// TwinCAT 3 PLC project PLC_MR
// ProgramVersion: 3.1.4026.16
// libraries:
//   Tc2_ControllerToolbox, * (Beckhoff Automation GmbH)
//   Tc2_SerialCom, * (Beckhoff Automation GmbH)
//   Tc2_Standard, * (Beckhoff Automation GmbH)
//   Tc2_System, * (Beckhoff Automation GmbH)
//   Tc2_Utilities, * (Beckhoff Automation GmbH)
//   Tc3_BA_Common, * (Beckhoff Automation GmbH)
//   Tc3_Module, * (Beckhoff Automation GmbH)
// project tree:
//   DUTs/ E_ControlMode.TcDUT, E_RampGeneratorState.TcDUT, E_RecipeRunETMode.TcDUT, E_RecipeRun.TcDUT, E_TowerLamp.TcDUT, OperationMode.TcDUT, outWord.TcDUT, RampGeneratorInput.TcDUT, RecipeRunET.TcDUT, RecipeStep.TcDUT, ScaleFactor.TcDUT (not stored)
//   FUNTION/ BOOL_TO_STRING_LHeaterON.TcPOU (not stored), CheckRangeSigned.TcPOU (not stored), CheckRangeUnsigned.TcPOU, HEXSTR_TO_REAL_LHeaterPV.TcPOU (not stored), Real_To_String_LineHeater.TcPOU, Real_To_String_ThermalBath.TcPOU, USINT_TO_WORD_Bit.TcPOU, WORD_TO_USINT_Bit.TcPOU
//   GVLs/ GVL_IO.TcGVL, GVL_Serial.TcGVL, RCP.TcGVL
//   / PlcTask.TcTTO (not stored), PlcTask_Standard.TcTTO
//   POUs/ FB_AnalogDeviceRampControl.TcPOU, FB_ControlRampGenerator.TcPOU, FB_DeviationCheck.TcPOU, FB_FaultCheck.TcPOU, FB_OverLimitCheck.TcPOU, FB_RecipeAnalogControlInputSequencer.TcPOU, FB_SensorLimitCheck.TcPOU, FB_TON_Pausable.TcPOU, FB_ValveControl.TcPOU, F_ResetTimersAndRCPTimes.TcPOU, MAIN.TcPOU, P11_E3508.TcPOU, P12_IQ_PLUS.TcPOU, P13_LineHeater.TcPOU, P14_ThermalBath.TcPOU, P15_RotationOperation.TcPOU, P16_CoverOperation.TcPOU, P17_DOROperation.TcPOU, P20_BackgroundCom.TcPOU (not stored), P21_Background_LineHeater.TcPOU, P22_Background_ThermalBath.TcPOU (not stored), P30_ManualControl.TcPOU, P50_RecipeControl.TcPOU, P60_UpdatePV.TcPOU, P70_Interface.TcPOU, P90_Interlock.TcPOU, P91_Monitoring.TcPOU, P92_Maintenance.TcPOU, P31_PriorityControl.TcPOU
// real-time tasks:
//   TASK PlcTask_Standard: cycle T#10ms, priority 21, ADS port 350
//   TASK PlcTask: cycle T#2ms, priority 19, ADS port 351
// I/O:
//   DEVICE Device 1 (EtherCAT) (disabled), AmsNetId 211.225.0.130.2.1
//     Term 1 (EK1200) [EK1200-5000 EtherCAT Power supply (2A E-Bus)]
//       Term 2 (EL6752) [EL6752 DeviceNet Master]
//       Term 3 (EL9011) [EL9011 End Terminal]
//   DEVICE Device 2 (EL6752) (disabled), AmsNetId 10.10.10.10.3.1
//     Box 1  (BK5220) // Bus Coupler
//     Box 2  (BK5220) // Bus Coupler
//     N4E0 1 // EDS-File: 'OPP6-2D.eds' DescText: OPP6-2D Vendor: CKD Corporation Device Type: Generic Device Product Name: OPP6-2D Catalog Number:
//     N4E0 2 // EDS-File: 'OPP6-2D.eds' DescText: OPP6-2D Vendor: CKD Corporation Device Type: Generic Device Product Name: OPP6-2D Catalog Number:
//     IQ-Plus // EDS-File: 'TBJQPDNG-L041X01 155Out154.eds' DescText: Intellisys IQ-Plus Vendor: Nor-Cal Products Device Type: Process Control Valve Product Name: INTELLISYS Catalog Number: IQ-Plus
//     E3508 // EDS-File: '3500-3.eds' DescText: Eurotherm 3500 Vendor: Eurotherm Device Type: Generic Product Name: Eurotherm 3500 Catalog Number:
//   DEVICE Device 3 (NOV-DP-RAM) (disabled)
// variable links:
//   PLC_MR/PLC_MR Instance <-> Device 2 (EL6752)/Box 1  (BK5220)
//     PlcTask_Standard Inputs/GVL_IO.aAnalogInputIO[1] <-> Term 15 (KL3464)/Channel 1/MFC01
//     PlcTask_Standard Inputs/GVL_IO.aAnalogInputIO[2] <-> Term 15 (KL3464)/Channel 2/MFC02
//     PlcTask_Standard Inputs/GVL_IO.aAnalogInputIO[3] <-> Term 15 (KL3464)/Channel 3/MFC03
//     PlcTask_Standard Inputs/GVL_IO.aAnalogInputIO[4] <-> Term 15 (KL3464)/Channel 4/MFC04
//     PlcTask_Standard Inputs/GVL_IO.aAnalogInputIO[5] <-> Term 17 (KL3464)/Channel 1/MFC05
//     PlcTask_Standard Inputs/GVL_IO.aAnalogInputIO[6] <-> Term 17 (KL3464)/Channel 2/MFC06
//     PlcTask_Standard Inputs/GVL_IO.aAnalogInputIO[7] <-> Term 17 (KL3464)/Channel 3/MFC07
//     PlcTask_Standard Inputs/GVL_IO.aAnalogInputIO[8] <-> Term 17 (KL3464)/Channel 4/MFC08
//     PlcTask_Standard Inputs/GVL_IO.aDigitalInputIO[{1..9}] <-> Term {2..10} (KL1408)/Channel 1/Input  (9 links)
//     PlcTask_Standard Inputs/GVL_IO.aDigitalInputIO[1] @bit 1 <-> Term 2 (KL1408)/Channel 2/Input
//     PlcTask_Standard Inputs/GVL_IO.aDigitalInputIO[1] @bit 2 <-> Term 2 (KL1408)/Channel 3/Input
//     PlcTask_Standard Inputs/GVL_IO.aDigitalInputIO[1] @bit 3 <-> Term 2 (KL1408)/Channel 4/Input
//     PlcTask_Standard Inputs/GVL_IO.aDigitalInputIO[1] @bit 4 <-> Term 2 (KL1408)/Channel 5/Input
//     PlcTask_Standard Inputs/GVL_IO.aDigitalInputIO[1] @bit 5 <-> Term 2 (KL1408)/Channel 6/Input
//     PlcTask_Standard Inputs/GVL_IO.aDigitalInputIO[1] @bit 6 <-> Term 2 (KL1408)/Channel 7/Input
//     PlcTask_Standard Inputs/GVL_IO.aDigitalInputIO[1] @bit 7 <-> Term 2 (KL1408)/Channel 8/Input
//     PlcTask_Standard Inputs/GVL_IO.aDigitalInputIO[2] @bit 1 <-> Term 3 (KL1408)/Channel 2/Input
//     PlcTask_Standard Inputs/GVL_IO.aDigitalInputIO[2] @bit 2 <-> Term 3 (KL1408)/Channel 3/Input
//     PlcTask_Standard Inputs/GVL_IO.aDigitalInputIO[2] @bit 3 <-> Term 3 (KL1408)/Channel 4/Input
//     PlcTask_Standard Inputs/GVL_IO.aDigitalInputIO[2] @bit 4 <-> Term 3 (KL1408)/Channel 5/Input
//     PlcTask_Standard Inputs/GVL_IO.aDigitalInputIO[2] @bit 5 <-> Term 3 (KL1408)/Channel 6/Input
//     PlcTask_Standard Inputs/GVL_IO.aDigitalInputIO[2] @bit 6 <-> Term 3 (KL1408)/Channel 7/Input
//     PlcTask_Standard Inputs/GVL_IO.aDigitalInputIO[2] @bit 7 <-> Term 3 (KL1408)/Channel 8/Input
//     PlcTask_Standard Inputs/GVL_IO.aDigitalInputIO[3] @bit 1 <-> Term 4 (KL1408)/Channel 2/Input
//     PlcTask_Standard Inputs/GVL_IO.aDigitalInputIO[3] @bit 2 <-> Term 4 (KL1408)/Channel 3/Input
//     PlcTask_Standard Inputs/GVL_IO.aDigitalInputIO[3] @bit 3 <-> Term 4 (KL1408)/Channel 4/Input
//     PlcTask_Standard Inputs/GVL_IO.aDigitalInputIO[3] @bit 4 <-> Term 4 (KL1408)/Channel 5/Input
//     PlcTask_Standard Inputs/GVL_IO.aDigitalInputIO[3] @bit 5 <-> Term 4 (KL1408)/Channel 6/Input
//     PlcTask_Standard Inputs/GVL_IO.aDigitalInputIO[3] @bit 6 <-> Term 4 (KL1408)/Channel 7/Input
//     PlcTask_Standard Inputs/GVL_IO.aDigitalInputIO[3] @bit 7 <-> Term 4 (KL1408)/Channel 8/Input
//     PlcTask_Standard Inputs/GVL_IO.aDigitalInputIO[4] @bit 1 <-> Term 5 (KL1408)/Channel 2/Input
//     PlcTask_Standard Inputs/GVL_IO.aDigitalInputIO[4] @bit 2 <-> Term 5 (KL1408)/Channel 3/Input
//     PlcTask_Standard Inputs/GVL_IO.aDigitalInputIO[4] @bit 3 <-> Term 5 (KL1408)/Channel 4/Input
//     PlcTask_Standard Inputs/GVL_IO.aDigitalInputIO[4] @bit 4 <-> Term 5 (KL1408)/Channel 5/Input
//     PlcTask_Standard Inputs/GVL_IO.aDigitalInputIO[4] @bit 5 <-> Term 5 (KL1408)/Channel 6/Input
//     PlcTask_Standard Inputs/GVL_IO.aDigitalInputIO[4] @bit 6 <-> Term 5 (KL1408)/Channel 7/Input
//     PlcTask_Standard Inputs/GVL_IO.aDigitalInputIO[4] @bit 7 <-> Term 5 (KL1408)/Channel 8/Input
//     PlcTask_Standard Inputs/GVL_IO.aDigitalInputIO[5] @bit 1 <-> Term 6 (KL1408)/Channel 2/Input
//     PlcTask_Standard Inputs/GVL_IO.aDigitalInputIO[5] @bit 2 <-> Term 6 (KL1408)/Channel 3/Input
//     PlcTask_Standard Inputs/GVL_IO.aDigitalInputIO[5] @bit 3 <-> Term 6 (KL1408)/Channel 4/Input
//     PlcTask_Standard Inputs/GVL_IO.aDigitalInputIO[5] @bit 4 <-> Term 6 (KL1408)/Channel 5/Input
//     PlcTask_Standard Inputs/GVL_IO.aDigitalInputIO[5] @bit 5 <-> Term 6 (KL1408)/Channel 6/Input
//     PlcTask_Standard Inputs/GVL_IO.aDigitalInputIO[5] @bit 6 <-> Term 6 (KL1408)/Channel 7/Input
//     PlcTask_Standard Inputs/GVL_IO.aDigitalInputIO[5] @bit 7 <-> Term 6 (KL1408)/Channel 8/Input
//     PlcTask_Standard Inputs/GVL_IO.aDigitalInputIO[6] @bit 1 <-> Term 7 (KL1408)/Channel 2/Input
//     PlcTask_Standard Inputs/GVL_IO.aDigitalInputIO[6] @bit 2 <-> Term 7 (KL1408)/Channel 3/Input
//     PlcTask_Standard Inputs/GVL_IO.aDigitalInputIO[6] @bit 3 <-> Term 7 (KL1408)/Channel 4/Input
//     PlcTask_Standard Inputs/GVL_IO.aDigitalInputIO[6] @bit 4 <-> Term 7 (KL1408)/Channel 5/Input
//     PlcTask_Standard Inputs/GVL_IO.aDigitalInputIO[6] @bit 5 <-> Term 7 (KL1408)/Channel 6/Input
//     PlcTask_Standard Inputs/GVL_IO.aDigitalInputIO[6] @bit 6 <-> Term 7 (KL1408)/Channel 7/Input
//     PlcTask_Standard Inputs/GVL_IO.aDigitalInputIO[6] @bit 7 <-> Term 7 (KL1408)/Channel 8/Input
//     PlcTask_Standard Inputs/GVL_IO.aDigitalInputIO[7] @bit 1 <-> Term 8 (KL1408)/Channel 2/Input
//     PlcTask_Standard Inputs/GVL_IO.aDigitalInputIO[7] @bit 2 <-> Term 8 (KL1408)/Channel 3/Input
//     PlcTask_Standard Inputs/GVL_IO.aDigitalInputIO[7] @bit 3 <-> Term 8 (KL1408)/Channel 4/Input
//     PlcTask_Standard Inputs/GVL_IO.aDigitalInputIO[7] @bit 4 <-> Term 8 (KL1408)/Channel 5/Input
//     PlcTask_Standard Inputs/GVL_IO.aDigitalInputIO[7] @bit 5 <-> Term 8 (KL1408)/Channel 6/Input
//     PlcTask_Standard Inputs/GVL_IO.aDigitalInputIO[7] @bit 6 <-> Term 8 (KL1408)/Channel 7/Input
//     PlcTask_Standard Inputs/GVL_IO.aDigitalInputIO[7] @bit 7 <-> Term 8 (KL1408)/Channel 8/Input
//     PlcTask_Standard Inputs/GVL_IO.aDigitalInputIO[8] @bit 1 <-> Term 9 (KL1408)/Channel 2/Input
//     PlcTask_Standard Inputs/GVL_IO.aDigitalInputIO[8] @bit 2 <-> Term 9 (KL1408)/Channel 3/Input
//     PlcTask_Standard Inputs/GVL_IO.aDigitalInputIO[8] @bit 3 <-> Term 9 (KL1408)/Channel 4/Input
//     PlcTask_Standard Inputs/GVL_IO.aDigitalInputIO[8] @bit 4 <-> Term 9 (KL1408)/Channel 5/Input
//     PlcTask_Standard Inputs/GVL_IO.aDigitalInputIO[8] @bit 5 <-> Term 9 (KL1408)/Channel 6/Input
//     PlcTask_Standard Inputs/GVL_IO.aDigitalInputIO[8] @bit 6 <-> Term 9 (KL1408)/Channel 7/Input
//     PlcTask_Standard Inputs/GVL_IO.aDigitalInputIO[8] @bit 7 <-> Term 9 (KL1408)/Channel 8/Input
//     PlcTask_Standard Inputs/GVL_IO.aDigitalInputIO[9] @bit 1 <-> Term 10 (KL1408)/Channel 2/Input
//     PlcTask_Standard Inputs/GVL_IO.aDigitalInputIO[9] @bit 2 <-> Term 10 (KL1408)/Channel 3/Input
//     PlcTask_Standard Inputs/GVL_IO.aDigitalInputIO[9] @bit 3 <-> Term 10 (KL1408)/Channel 4/Input
//     PlcTask_Standard Inputs/GVL_IO.aDigitalInputIO[9] @bit 4 <-> Term 10 (KL1408)/Channel 5/Input
//     PlcTask_Standard Inputs/GVL_IO.aDigitalInputIO[9] @bit 5 <-> Term 10 (KL1408)/Channel 6/Input
//     PlcTask_Standard Inputs/GVL_IO.aDigitalInputIO[9] @bit 6 <-> Term 10 (KL1408)/Channel 7/Input
//     PlcTask_Standard Inputs/GVL_IO.aDigitalInputIO[9] @bit 7 <-> Term 10 (KL1408)/Channel 8/Input
//     PlcTask_Standard Outputs/GVL_IO.aAnalogOutputIO[1] <-> Term 16 (KL4404)/Channel 1/MFC01
//     PlcTask_Standard Outputs/GVL_IO.aAnalogOutputIO[2] <-> Term 16 (KL4404)/Channel 2/MFC02
//     PlcTask_Standard Outputs/GVL_IO.aAnalogOutputIO[3] <-> Term 16 (KL4404)/Channel 3/MFC03
//     PlcTask_Standard Outputs/GVL_IO.aAnalogOutputIO[4] <-> Term 16 (KL4404)/Channel 4/MFC04
//     PlcTask_Standard Outputs/GVL_IO.aAnalogOutputIO[5] <-> Term 18 (KL4404)/Channel 1/MFC05
//     PlcTask_Standard Outputs/GVL_IO.aAnalogOutputIO[6] <-> Term 18 (KL4404)/Channel 2/MFC06
//     PlcTask_Standard Outputs/GVL_IO.aAnalogOutputIO[7] <-> Term 18 (KL4404)/Channel 3/MFC07
//     PlcTask_Standard Outputs/GVL_IO.aAnalogOutputIO[8] <-> Term 18 (KL4404)/Channel 4/MFC08
//     PlcTask_Standard Outputs/GVL_IO.aDigitalOutputIO[{1..4}] <-> Term {11..14} (KL2408)/Channel 1/Output  (4 links)
//     PlcTask_Standard Outputs/GVL_IO.aDigitalOutputIO[1] @bit 1 <-> Term 11 (KL2408)/Channel 2/Output
//     PlcTask_Standard Outputs/GVL_IO.aDigitalOutputIO[1] @bit 2 <-> Term 11 (KL2408)/Channel 3/Output
//     PlcTask_Standard Outputs/GVL_IO.aDigitalOutputIO[1] @bit 3 <-> Term 11 (KL2408)/Channel 4/Output
//     PlcTask_Standard Outputs/GVL_IO.aDigitalOutputIO[1] @bit 4 <-> Term 11 (KL2408)/Channel 5/Output
//     PlcTask_Standard Outputs/GVL_IO.aDigitalOutputIO[1] @bit 5 <-> Term 11 (KL2408)/Channel 6/Output
//     PlcTask_Standard Outputs/GVL_IO.aDigitalOutputIO[1] @bit 6 <-> Term 11 (KL2408)/Channel 7/Output
//     PlcTask_Standard Outputs/GVL_IO.aDigitalOutputIO[1] @bit 7 <-> Term 11 (KL2408)/Channel 8/Output
//     PlcTask_Standard Outputs/GVL_IO.aDigitalOutputIO[2] @bit 1 <-> Term 12 (KL2408)/Channel 2/Output
//     PlcTask_Standard Outputs/GVL_IO.aDigitalOutputIO[2] @bit 2 <-> Term 12 (KL2408)/Channel 3/Output
//     PlcTask_Standard Outputs/GVL_IO.aDigitalOutputIO[2] @bit 3 <-> Term 12 (KL2408)/Channel 4/Output
//     PlcTask_Standard Outputs/GVL_IO.aDigitalOutputIO[2] @bit 4 <-> Term 12 (KL2408)/Channel 5/Output
//     PlcTask_Standard Outputs/GVL_IO.aDigitalOutputIO[2] @bit 5 <-> Term 12 (KL2408)/Channel 6/Output
//     PlcTask_Standard Outputs/GVL_IO.aDigitalOutputIO[2] @bit 6 <-> Term 12 (KL2408)/Channel 7/Output
//     PlcTask_Standard Outputs/GVL_IO.aDigitalOutputIO[2] @bit 7 <-> Term 12 (KL2408)/Channel 8/Output
//     PlcTask_Standard Outputs/GVL_IO.aDigitalOutputIO[3] @bit 1 <-> Term 13 (KL2408)/Channel 2/Output
//     PlcTask_Standard Outputs/GVL_IO.aDigitalOutputIO[3] @bit 2 <-> Term 13 (KL2408)/Channel 3/Output
//     PlcTask_Standard Outputs/GVL_IO.aDigitalOutputIO[3] @bit 3 <-> Term 13 (KL2408)/Channel 4/Output
//     PlcTask_Standard Outputs/GVL_IO.aDigitalOutputIO[3] @bit 4 <-> Term 13 (KL2408)/Channel 5/Output
//     PlcTask_Standard Outputs/GVL_IO.aDigitalOutputIO[3] @bit 5 <-> Term 13 (KL2408)/Channel 6/Output
//     PlcTask_Standard Outputs/GVL_IO.aDigitalOutputIO[3] @bit 6 <-> Term 13 (KL2408)/Channel 7/Output
//     PlcTask_Standard Outputs/GVL_IO.aDigitalOutputIO[3] @bit 7 <-> Term 13 (KL2408)/Channel 8/Output
//     PlcTask_Standard Outputs/GVL_IO.aDigitalOutputIO[4] @bit 1 <-> Term 14 (KL2408)/Channel 2/Output
//     PlcTask_Standard Outputs/GVL_IO.aDigitalOutputIO[4] @bit 2 <-> Term 14 (KL2408)/Channel 3/Output
//     PlcTask_Standard Outputs/GVL_IO.aDigitalOutputIO[4] @bit 3 <-> Term 14 (KL2408)/Channel 4/Output
//     PlcTask_Standard Outputs/GVL_IO.aDigitalOutputIO[4] @bit 4 <-> Term 14 (KL2408)/Channel 5/Output
//     PlcTask_Standard Outputs/GVL_IO.aDigitalOutputIO[4] @bit 5 <-> Term 14 (KL2408)/Channel 6/Output
//     PlcTask_Standard Outputs/GVL_IO.aDigitalOutputIO[4] @bit 6 <-> Term 14 (KL2408)/Channel 7/Output
//     PlcTask_Standard Outputs/GVL_IO.aDigitalOutputIO[4] @bit 7 <-> Term 14 (KL2408)/Channel 8/Output
//   PLC_MR/PLC_MR Instance <-> Device 2 (EL6752)/Box 2  (BK5220)
//     PlcTask Inputs/P21_Background_LineHeater.stIn_KL6031_LH/D <-> Term 34 (KL6031)/Channel 1/Data In 0
//     PlcTask Inputs/P21_Background_LineHeater.stIn_KL6031_LH/D @bit {8..168 step 8} <-> Term 34 (KL6031)/Channel 1/Data In {1..21}  (21 links)
//     PlcTask Inputs/P21_Background_LineHeater.stIn_KL6031_LH/Status <-> Term 34 (KL6031)/Channel 1/State
//     PlcTask Inputs/P22_Background_ThermalBath.stIn_KL6031_TB/D <-> Term 35 (KL6031)/Channel 1/Data In 0
//     PlcTask Inputs/P22_Background_ThermalBath.stIn_KL6031_TB/D @bit {8..168 step 8} <-> Term 35 (KL6031)/Channel 1/Data In {1..21}  (21 links)
//     PlcTask Inputs/P22_Background_ThermalBath.stIn_KL6031_TB/Status <-> Term 35 (KL6031)/Channel 1/State
//     PlcTask Outputs/P21_Background_LineHeater.stOut_KL6031_LH/Ctrl <-> Term 34 (KL6031)/Channel 1/Ctrl
//     PlcTask Outputs/P21_Background_LineHeater.stOut_KL6031_LH/D <-> Term 34 (KL6031)/Channel 1/Data Out 0
//     PlcTask Outputs/P21_Background_LineHeater.stOut_KL6031_LH/D @bit {8..168 step 8} <-> Term 34 (KL6031)/Channel 1/Data Out {1..21}  (21 links)
//     PlcTask Outputs/P22_Background_ThermalBath.stOut_KL6031_TB/Ctrl <-> Term 35 (KL6031)/Channel 1/Ctrl
//     PlcTask Outputs/P22_Background_ThermalBath.stOut_KL6031_TB/D <-> Term 35 (KL6031)/Channel 1/Data Out 0
//     PlcTask Outputs/P22_Background_ThermalBath.stOut_KL6031_TB/D @bit {8..168 step 8} <-> Term 35 (KL6031)/Channel 1/Data Out {1..21}  (21 links)
//     PlcTask_Standard Inputs/GVL_IO.aAnalogInputIO2[1] <-> Term 32 (KL3152)/Channel 1/RotaionPV
//     PlcTask_Standard Inputs/GVL_IO.aAnalogInputIO[10] <-> Term 20 (KL3464)/Channel 2/MFC10
//     PlcTask_Standard Inputs/GVL_IO.aAnalogInputIO[11] <-> Term 20 (KL3464)/Channel 3/MFC11
//     PlcTask_Standard Inputs/GVL_IO.aAnalogInputIO[12] <-> Term 20 (KL3464)/Channel 4/MFC12
//     PlcTask_Standard Inputs/GVL_IO.aAnalogInputIO[13] <-> Term 22 (KL3464)/Channel 1/MFC13
//     PlcTask_Standard Inputs/GVL_IO.aAnalogInputIO[14] <-> Term 22 (KL3464)/Channel 2/MFC14
//     PlcTask_Standard Inputs/GVL_IO.aAnalogInputIO[15] <-> Term 22 (KL3464)/Channel 3/MFC15
//     PlcTask_Standard Inputs/GVL_IO.aAnalogInputIO[16] <-> Term 22 (KL3464)/Channel 4/MFC16
//     PlcTask_Standard Inputs/GVL_IO.aAnalogInputIO[17] <-> Term 24 (KL3464)/Channel 1/MFC17
//     PlcTask_Standard Inputs/GVL_IO.aAnalogInputIO[18] <-> Term 24 (KL3464)/Channel 2/MFC18
//     PlcTask_Standard Inputs/GVL_IO.aAnalogInputIO[19] <-> Term 24 (KL3464)/Channel 3/MFC19
//     PlcTask_Standard Inputs/GVL_IO.aAnalogInputIO[9] <-> Term 20 (KL3464)/Channel 1/MFC09
//     PlcTask_Standard Inputs/GVL_IO.aAnalogInputIO[20] <-> Term 24 (KL3464)/Channel 4/EPC01
//     PlcTask_Standard Inputs/GVL_IO.aAnalogInputIO[21] <-> Term 26 (KL3464)/Channel 1/EPC02
//     PlcTask_Standard Inputs/GVL_IO.aAnalogInputIO[22] <-> Term 26 (KL3464)/Channel 2/EPC03
//     PlcTask_Standard Inputs/GVL_IO.aAnalogInputIO[23] <-> Term 26 (KL3464)/Channel 3/EPC04
//     PlcTask_Standard Inputs/GVL_IO.aAnalogInputIO[24] <-> Term 26 (KL3464)/Channel 4/EPC05
//     PlcTask_Standard Inputs/GVL_IO.aAnalogInputIO[25] <-> Term 28 (KL3464)/Channel 1/EPC06
//     PlcTask_Standard Inputs/GVL_IO.aAnalogInputIO[26] <-> Term 28 (KL3464)/Channel 2/EPC07
//     PlcTask_Standard Inputs/GVL_IO.aAnalogInputIO[27] <-> Term 28 (KL3464)/Channel 3/UPressure
//     PlcTask_Standard Inputs/GVL_IO.aAnalogInputIO[28] <-> Term 28 (KL3464)/Channel 4/ExPressure
//     PlcTask_Standard Inputs/GVL_IO.aAnalogInputIO[29] <-> Term 30 (KL3464)/Channel 1/Data
//     PlcTask_Standard Inputs/GVL_IO.aAnalogInputIO[37] <-> Term 33 (KL3204)/Channel 1/Data
//     PlcTask_Standard Inputs/GVL_IO.aAnalogInputIO[38] <-> Term 33 (KL3204)/Channel 2/Data
//     PlcTask_Standard Inputs/GVL_IO.aAnalogInputIO[33] <-> Term 31 (KL3054)/Channel 1/S01
//     PlcTask_Standard Inputs/GVL_IO.aAnalogInputIO[34] <-> Term 31 (KL3054)/Channel 2/S02
//     PlcTask_Standard Inputs/GVL_IO.aAnalogInputIO[35] <-> Term 31 (KL3054)/Channel 3/S03
//     PlcTask_Standard Inputs/GVL_IO.aAnalogInputIO[36] <-> Term 31 (KL3054)/Channel 4/S04
//     PlcTask_Standard Outputs/GVL_IO.aAnalogOutputIO[10] <-> Term 21 (KL4404)/Channel 2/MFC10
//     PlcTask_Standard Outputs/GVL_IO.aAnalogOutputIO[11] <-> Term 21 (KL4404)/Channel 3/MFC11
//     PlcTask_Standard Outputs/GVL_IO.aAnalogOutputIO[12] <-> Term 21 (KL4404)/Channel 4/MFC12
//     PlcTask_Standard Outputs/GVL_IO.aAnalogOutputIO[13] <-> Term 23 (KL4404)/Channel 1/MFC13
//     PlcTask_Standard Outputs/GVL_IO.aAnalogOutputIO[14] <-> Term 23 (KL4404)/Channel 2/MFC14
//     PlcTask_Standard Outputs/GVL_IO.aAnalogOutputIO[15] <-> Term 23 (KL4404)/Channel 3/MFC15
//     PlcTask_Standard Outputs/GVL_IO.aAnalogOutputIO[16] <-> Term 23 (KL4404)/Channel 4/MFC16
//     PlcTask_Standard Outputs/GVL_IO.aAnalogOutputIO[17] <-> Term 25 (KL4404)/Channel 1/MFC17
//     PlcTask_Standard Outputs/GVL_IO.aAnalogOutputIO[18] <-> Term 25 (KL4404)/Channel 2/MFC18
//     PlcTask_Standard Outputs/GVL_IO.aAnalogOutputIO[19] <-> Term 25 (KL4404)/Channel 3/MFC19
//     PlcTask_Standard Outputs/GVL_IO.aAnalogOutputIO[9] <-> Term 21 (KL4404)/Channel 1/MFC09
//     PlcTask_Standard Outputs/GVL_IO.aAnalogOutputIO[20] <-> Term 25 (KL4404)/Channel 4/EPC01
//     PlcTask_Standard Outputs/GVL_IO.aAnalogOutputIO[21] <-> Term 27 (KL4404)/Channel 1/EPC02
//     PlcTask_Standard Outputs/GVL_IO.aAnalogOutputIO[22] <-> Term 27 (KL4404)/Channel 2/EPC03
//     PlcTask_Standard Outputs/GVL_IO.aAnalogOutputIO[23] <-> Term 27 (KL4404)/Channel 3/EPC04
//     PlcTask_Standard Outputs/GVL_IO.aAnalogOutputIO[24] <-> Term 27 (KL4404)/Channel 4/EPC05
//     PlcTask_Standard Outputs/GVL_IO.aAnalogOutputIO[25] <-> Term 29 (KL4404)/Channel 1/EPC06
//     PlcTask_Standard Outputs/GVL_IO.aAnalogOutputIO[26] <-> Term 29 (KL4404)/Channel 2/EPC07
//     PlcTask_Standard Outputs/GVL_IO.aAnalogOutputIO[27] <-> Term 29 (KL4404)/Channel 3/ExPressure
//     PlcTask_Standard Outputs/GVL_IO.aAnalogOutputIO[28] <-> Term 29 (KL4404)/Channel 4/RotationSV
//   PLC_MR/PLC_MR Instance <-> Device 2 (EL6752)/E3508
//     PlcTask_Standard Inputs/P11_E3508.aInputCVBytes[1] <-> Connection (Poll)/Inputs/Input Data_7
//     PlcTask_Standard Inputs/P11_E3508.aInputCVBytes[2] <-> Connection (Poll)/Inputs/Input Data_8
//     PlcTask_Standard Inputs/P11_E3508.aInputDerivative[1] <-> Connection (Poll)/Inputs/Input Data_19
//     PlcTask_Standard Inputs/P11_E3508.aInputDerivative[2] <-> Connection (Poll)/Inputs/Input Data_20
//     PlcTask_Standard Inputs/P11_E3508.aInputIntegral[1] <-> Connection (Poll)/Inputs/Input Data_17
//     PlcTask_Standard Inputs/P11_E3508.aInputIntegral[2] <-> Connection (Poll)/Inputs/Input Data_18
//     PlcTask_Standard Inputs/P11_E3508.aInputPVBytes[1] <-> Connection (Poll)/Inputs/Input Data_1
//     PlcTask_Standard Inputs/P11_E3508.aInputPVBytes[2] <-> Connection (Poll)/Inputs/Input Data_2
//     PlcTask_Standard Inputs/P11_E3508.aInputProportional[1] <-> Connection (Poll)/Inputs/Input Data_15
//     PlcTask_Standard Inputs/P11_E3508.aInputProportional[2] <-> Connection (Poll)/Inputs/Input Data_16
//     PlcTask_Standard Inputs/P11_E3508.aInputSVBytes[1] <-> Connection (Poll)/Inputs/Input Data_3
//     PlcTask_Standard Inputs/P11_E3508.aInputSVBytes[2] <-> Connection (Poll)/Inputs/Input Data_4
//     PlcTask_Standard Inputs/P11_E3508.aInputTVBytes[1] <-> Connection (Poll)/Inputs/Input Data_5
//     PlcTask_Standard Inputs/P11_E3508.aInputTVBytes[2] <-> Connection (Poll)/Inputs/Input Data_6
//     PlcTask_Standard Inputs/P11_E3508.nInputAlarmBytes <-> Connection (Poll)/Inputs/Input Data_9
//     PlcTask_Standard Inputs/P11_E3508.nInputManAutoBytes <-> Connection (Poll)/Inputs/Input Data_11
//     PlcTask_Standard Outputs/P11_E3508.aOutputPowerBytes[1] <-> Connection (Poll)/Outputs/Output Data_5
//     PlcTask_Standard Outputs/P11_E3508.aOutputPowerBytes[2] <-> Connection (Poll)/Outputs/Output Data_6
//     PlcTask_Standard Outputs/P11_E3508.aOutputSVBytes[1] <-> Connection (Poll)/Outputs/Output Data_1
//     PlcTask_Standard Outputs/P11_E3508.aOutputSVBytes[2] <-> Connection (Poll)/Outputs/Output Data_2
//     PlcTask_Standard Outputs/P11_E3508.nOutputManAutoBytes <-> Connection (Poll)/Outputs/Output Data_3
//   PLC_MR/PLC_MR Instance <-> Device 2 (EL6752)/IQ-Plus
//     PlcTask_Standard Inputs/P12_IQ_PLUS.aInputPressurePV_CDG1[1] <-> Connection (Poll)/Inputs/Input 155_2
//     PlcTask_Standard Inputs/P12_IQ_PLUS.aInputPressurePV_CDG1[2] <-> Connection (Poll)/Inputs/Input 155_3
//     PlcTask_Standard Inputs/P12_IQ_PLUS.aInputPressurePV_CDG2[1] <-> Connection (Poll)/Inputs/Input 155_4
//     PlcTask_Standard Inputs/P12_IQ_PLUS.aInputPressurePV_CDG2[2] <-> Connection (Poll)/Inputs/Input 155_5
//     PlcTask_Standard Inputs/P12_IQ_PLUS.aInputPressureSP[1] <-> Connection (Poll)/Inputs/Input 155_6
//     PlcTask_Standard Inputs/P12_IQ_PLUS.aInputPressureSP[2] <-> Connection (Poll)/Inputs/Input 155_7
//     PlcTask_Standard Inputs/P12_IQ_PLUS.aInputValvePosionPV[1] <-> Connection (Poll)/Inputs/Input 155_8
//     PlcTask_Standard Inputs/P12_IQ_PLUS.aInputValvePosionPV[2] <-> Connection (Poll)/Inputs/Input 155_9
//     PlcTask_Standard Inputs/P12_IQ_PLUS.nInputStatus <-> Connection (Poll)/Inputs/Input 155_1
//     PlcTask_Standard Outputs/P12_IQ_PLUS.aOutputSVBytes[1] <-> Connection (Poll)/Outputs/Output 154[1]
//     PlcTask_Standard Outputs/P12_IQ_PLUS.aOutputSVBytes[2] <-> Connection (Poll)/Outputs/Output 154[2]
//     PlcTask_Standard Outputs/P12_IQ_PLUS.nOutputMode <-> Connection (Poll)/Outputs/Output 154[0]
//     PlcTask_Standard Outputs/P12_IQ_PLUS.nOutputSetType <-> Connection (Poll)/Outputs/Output 154[3]
//   PLC_MR/PLC_MR Instance <-> Device 2 (EL6752)/N4E0 1
//     PlcTask_Standard Outputs/GVL_IO.aOutputSolValve[1] <-> Connection (Poll)/Outputs/Output Data
//   PLC_MR/PLC_MR Instance <-> Device 2 (EL6752)/N4E0 2
//     PlcTask_Standard Outputs/GVL_IO.aOutputSolValve[2] <-> Connection (Poll)/Outputs/Output Data

CONFIGURATION PLC_MR
    RESOURCE PLC ON TwinCAT3
        TASK PlcTask_Standard(INTERVAL := T#10ms, PRIORITY := 21);
        PROGRAM MAIN WITH PlcTask_Standard : MAIN;
    END_RESOURCE
END_CONFIGURATION

// ---- DUTs/E_ControlMode.TcDUT
{attribute 'qualified_only'}
{attribute 'strict'}
{attribute 'to_string'}
TYPE E_ControlMode :
(
	Manual := 0,
	Recipe := 1,
	Priority := 2
);
END_TYPE

// ---- DUTs/E_RampGeneratorState.TcDUT
{attribute 'qualified_only'}
{attribute 'strict'}
{attribute 'to_string'}
TYPE E_RampGeneratorState :
(
	Init := 0,
	Run := 1,
	End := 2
);
END_TYPE

// ---- DUTs/E_RecipeRunETMode.TcDUT
{attribute 'qualified_only'}
{attribute 'strict'}
{attribute 'to_string'}
TYPE E_RecipeRunETMode :
(
	None := 0,
	Ramp := 1,
	Hold := 2
);
END_TYPE

// ---- DUTs/E_RecipeRun.TcDUT
{attribute 'qualified_only'}
{attribute 'strict'}
{attribute 'to_string'}
TYPE E_RecipeRun :
(
	Initial := 1,		// 초기화 상태 (변수 초기화)
	Ramp := 2,			// Ramp 처리 상태 (현재 스텝의 동작 수행)
	CheckHoldTemp := 3,	// Hold Type 확인
	End := 5
);
END_TYPE

// ---- DUTs/E_TowerLamp.TcDUT
{attribute 'qualified_only'}
{attribute 'strict'}
{attribute 'to_string'}
TYPE E_TowerLamp :
(
	OFF, //대기상태 (Signal)
	RED, // Alarm
	YELLOW, // Warning
	GREEN, // Running
	BLUE, // Maint
	WHITE, // Idle
	BUZZER
):= OFF;
END_TYPE

// ---- DUTs/OperationMode.TcDUT
{attribute 'qualified_only'}
{attribute 'strict'}
{attribute 'to_string'}
TYPE OperationMode :
(
	Manual := 0,
	Recipe := 1,
	Emergency := 2
);
END_TYPE

// ---- DUTs/outWord.TcDUT
TYPE outWord :
STRUCT
	Lower : USINT; //Lower Bytes
	Upper : USINT; //Upper Bytes
END_STRUCT
END_TYPE

// ---- DUTs/RampGeneratorInput.TcDUT
TYPE RampGeneratorInput :
STRUCT
	restart : BOOL;
	targetValue : REAL;
	rampTime : UINT := 1;
END_STRUCT
END_TYPE

// ---- DUTs/RecipeRunET.TcDUT
TYPE RecipeRunET :
STRUCT
	ET : TIME := T#0S;
	Mode: E_RecipeRunETMode := E_RecipeRunETMode.None;
END_STRUCT
END_TYPE

// ---- DUTs/RecipeStep.TcDUT
TYPE RecipeStep :
STRUCT
	sRecipe : STRING(81);
	iRecipe : ARRAY[1..9] OF INT; //Reactor Condition
	rRecipe : ARRAY[1..26] OF REAL; //MFC, EPC Data
	dRecipe : DWORD; //Valve Data
END_STRUCT
END_TYPE

// ---- GVLs/GVL_IO.TcGVL
{attribute 'qualified_only'}
VAR_GLOBAL
	(* Digital IO to Byte *)
	aDigitalInputIO AT %I* 	: ARRAY[1..9]OF BYTE; //KL1408 9EA
	aDigitalOutputIO AT %Q* : ARRAY[1..4]OF BYTE; //KL2408 4EA
	
	(* Analog Input to INT*)
	aAnalogInputIO AT %I* 	: ARRAY[1..40]OF INT;
	aAnalogOutputIO AT %Q* 	: ARRAY[1..NumAnalogController ] OF INT;
	aAnalogInputIO2 AT %I*	: ARRAY[1..2]OF UINT;
	
	(*Solenoid Valve*)
	aOutputSolValve AT %Q* 	: ARRAY[1..3]OF DWORD; //Solenoid Valve
	
	(* Read and Write of Device Control Value*)
	aController 			: ARRAY[1..NumAnalogController] OF FB_ControlRampGenerator; //MFC, EPC 0 ~ 5V
	aController_PV 			: ARRAY[1..NumAnalogController] OF REAL; //Present Value from Device
	aReactorMaxValue		: ARRAY[1..NumReactor] OF REAL;
	
	(* Present Value Meter Display*)
	aMonitoring_PV 			: ARRAY[1..17] OF REAL; //Gauge Monitoring Value to UI
	aInputState				: ARRAY[1..5] OF WORD; // Digital Input from Device (Switch)
	aOutputCmd				: ARRAY[1..3] OF WORD; // Digital Command from UI
	aInterlock				: ARRAY[1..5] OF DWORD; // Interlock
	aInterlockSet			: ARRAY[1..16] OF REAL; // UI Interlokc Setting Value
	aInterlockEnable		: ARRAY[1..6] OF DWORD; // UI Interlock Enable Setting
	
	nCaseSignalTower		: INT;
	nDorOperationError		: INT;
	bDorState				: BOOL;
	bDorOnEnable			: BOOL;
// 	bE3508_HeaterOn			: BOOL;
	wE3508_PV				: WORD;
	wIqPlus_CDG1_PV			: WORD;
	wIqPlus_CDG2_PV			: WORD;
	nRotation_Converted_PV	: INT;
	nIQPLUS_SetType 		: INT;
	nIQPLUS_Mode			: INT;
	tRecipeControl_Ramp_ET	: TIME;
	tRecipeControl_Hold_ET	: TIME;
	tRecipeControl_Pause_ET	: TIME;
	aLineHeater_rTemperaturePV : ARRAY[1..8]OF REAL;
	nE3508_nInputManAutoBytes : USINT;
	isCoverClosed 			: BOOL;
	isPumpRunning 			: BOOL;
	
	nUIInterockCheckOpenReactor : WORD;
	nUIInterockCheckRecipeEnable : WORD;
END_VAR

VAR_GLOBAL CONSTANT
	KL3464MaxValueH	: REAL := 16383; //0~5V Half Input
	KL3464MaxValue 	: REAL := 32767; //0~10V
	KL4404MaxValueH	: REAL := 16383; //0~5V Half Output
	KL3054MaxValue 	: REAL := 32767; //4~20mA
	KL3152MaxValue	: REAL := 65535; //4~20mA
	KL3204MaxValue 	: REAL := 32767; //4~20mA
	
	NumAnalogController : UINT := 29;
	NumFlowController : UINT := 26;
	NumReactor : UINT := 3;
	
	AnalogControllerOutputVoltage : REAL := 5;
	TempDigitOutputFallbackThres : REAL := 10;
END_VAR

// ---- GVLs/GVL_Serial.TcGVL
//{attribute 'qualified_only'}
VAR_GLOBAL
	TxBufferTB : ComBuffer; (* Receive data buffer; used with all receive function blocks *)
	RxBufferTB : ComBuffer; (* Transmit data buffer; used with all receive function blocks *)
	
	TxBufferLH : ComBuffer; //잘동작되면 TB도 지역변수로 변경
	RxBufferLH : ComBuffer;	
END_VAR

// ---- GVLs/RCP.TcGVL
{attribute 'qualified_only'}
VAR_GLOBAL
	aRecipe		: ARRAY[1..100] OF RecipeStep; //Recipe Structure
	iRcpTotalStep			: INT; //Recip Total Number
	
	iRcpStepN				: INT;
	cmd_RcpOperation		: INT; // 0:Inital State, 10:RUN, 20:PAUSE, 30:RESTART, 40:STOP, 60:SKIP, 90:ManualOperation
	userState				: INT;	// 0:Inital State, 10:RUN, 20:PAUSE, 30:RESTART, 40:STOP, 50:END, 60:SKIP
	
	Pause_ET				: TIME := T#0S;
	RecipeRunET 			: RecipeRunET; 
	TotalET				: TIME := T#0S;
END_VAR

// ---- POUs/MAIN.TcPOU
PROGRAM MAIN
VAR_INPUT
	controlModeCmd : E_ControlMode := E_ControlMode.Manual;
END_VAR
VAR
	controlMode	: E_ControlMode := controlModeCmd;
	prevControlMode : E_ControlMode := controlMode;
END_VAR

(* Modify Program *)

P11_E3508(); //Temp Controller
P12_IQ_PLUS(); //Throttle Valve Controller
P13_LineHeater();
P14_ThermalBath();
P15_RotationOperation();
P16_CoverOperation();
P17_DOROperation();
P20_BackgroundCom();
P21_Background_LineHeater();
P22_Background_ThermalBath();
P22_Background_ThermalBath();


IF controlMode <> E_ControlMode.Priority THEN
	IF controlMode <> controlModeCmd THEN
		IF controlModeCmd = E_ControlMode.Priority THEN
			prevControlMode := controlMode;
		END_IF
		controlMode := controlModeCmd;
	END_IF
END_IF

CASE controlMode OF
	E_ControlMode.Manual:
		P30_ManualControl();
	
	E_ControlMode.Recipe:
		P50_RecipeControl(); //레시피 콘트론
		
	E_ControlMode.Priority:
		P31_PriorityControl();
		IF P31_PriorityControl.complete = TRUE THEN
			controlMode := prevControlMode;
			controlModeCmd := controlMode;
		END_IF
END_CASE

P60_UpdatePV();
P70_Interface();
P90_Interlock();
P91_Monitoring();
P92_Maintenance();
(* Interlock Condtion *)
// DOR Operation Condition

END_PROGRAM

// ---- POUs/P11_E3508.TcPOU
PROGRAM P11_E3508
VAR
	wControlValue			: WORD;
	wPowerRateSetValue		: WORD;	
	bOutputManAuto 			: BOOL; // Command 0:Auto, 1:Manual Mode
	
	bHeaterOn				: BOOL := FALSE; //to PSTEK
	bHeaterReset			: BOOL; //to PSTEK

	bAlarmState_E3508 		: BOOL; //Alarm or Sensor Break Signal
	bManAuto_E3508 			: BOOL; //State, 0:Manual, 1:Auto

	isHeaterReady			: BOOL; //Close : Ready
	isHeaterRun				: BOOL; //Close : Running, Open : Stop
	isHeaterFault			: BOOL; //Close : Falut, Open : Normal
	//isInductionHeaterErr	: BOOL; //Power Supply
	bInductionHeaterCB		: BOOL;
	//Input from E3508 Controller
	aInputPVBytes AT %I* 		: ARRAY[1..2]OF USINT; //Input Process Values
	aInputSVBytes AT %I* 		: ARRAY[1..2]OF USINT; //Input Set Values
	aInputTVBytes AT %I* 		: ARRAY[1..2]OF USINT; //Input Target Valuse
	aInputCVBytes AT %I* 		: ARRAY[1..2]OF USINT; //Induction Heter Controlled Values
	aInputProportional AT %I* 	: ARRAY[1..2]OF USINT; //PID - Proportional Band
	aInputIntegral AT %I* 		: ARRAY[1..2]OF USINT; //PID - Integral Time
	aInputDerivative AT %I* 	: ARRAY[1..2]OF USINT; //PID - Derivative Time 
	nInputAlarmBytes AT %I* 	: USINT; // Alarm State
	nInputManAutoBytes AT %I* 	: USINT; // ManAuto State
	
	wE3508_PV				: WORD;
	wE3508_SV				: WORD;
	wE3508_PowerRate		: WORD; //To Induction Heater Control Values
	wE3508_P				: WORD; //PID Parameter P
	wE3508_I				: WORD; //PID Parameter I
	wE3508_D				: WORD; //PID Parameter D
	//Output to E3508 Controller
	wOutputSVBytes 				: outWord;
	wOutputPowerSVBytes 		: outWord;
	aOutputSVBytes AT %Q* 		: ARRAY[1..2]OF USINT; //Temperature Set Value
	nOutputManAutoBytes AT %Q* 	: USINT; //ManAuto Change
	aOutputPowerBytes AT %Q* 	: ARRAY[1..2]OF USINT; //Output Power in Manual State
	//nOutputAlarmClear AT %Q* : USINT; //Alarm Clear Set
END_VAR

//Induction Heater & Temperature Controller & Thermo Couple(R-Type)
//Maker: PSTEK, Eurotherm
//Model: 3508
//Temperature Range: 0 ~ 12000℃

(* Command *)
bHeaterOn := GVL_IO.aOutputCmd[1].4;
bHeaterReset := GVL_IO.aOutputCmd[1].5;
nOutputManAutoBytes.0 := GVL_IO.aOutputCmd[1].11; //Temp Controller Mode Command

(* Read from Power Distribution Pannel *)
bInductionHeaterCB		:= GVL_IO.aDigitalInputIO[4].7;
nInputAlarmBytes.7 		:= GVL_IO.aInputState[4].7;
nInputManAutoBytes.7 	:= GVL_IO.aInputState[4].8;

(* Read from E3508 Device Value *)
wE3508_PV				:= USINT_TO_WORD_Bit(aInputPVBytes[1], aInputPVBytes[2]);
wE3508_SV				:= USINT_TO_WORD_Bit(aInputSVBytes[1], aInputSVBytes[2]);
wE3508_PowerRate		:= USINT_TO_WORD_Bit(aInputCVBytes[1], aInputCVBytes[2]); //divided to 10
wE3508_P 				:= USINT_TO_WORD_Bit(aInputProportional[1], aInputProportional[2]);
wE3508_I 				:= USINT_TO_WORD_Bit(aInputIntegral[1], aInputIntegral[2]);
wE3508_D 				:= USINT_TO_WORD_Bit(aInputDerivative[1], aInputDerivative[2]);

//bAlarmState_E3508 		:= nInputAlarmBytes.7;

GVL_IO.aMonitoring_PV[10] := WORD_TO_REAL(wE3508_PowerRate)*0.1; //divided to 10 PowerRate

(* Read from Induction Heater Value *)
isHeaterReady 			:= GVL_IO.aDigitalInputIO[2].2;
isHeaterRun		 		:= GVL_IO.aDigitalInputIO[2].3;
isHeaterFault 			:= GVL_IO.aDigitalInputIO[2].4;

// Interface with other PRGs
wControlValue			:= LREAL_TO_WORD(GVL_IO.aController[27].rControlValue);
GVL_IO.wE3508_PV		:= wE3508_PV;

(* Write to E3508 Device Value *)
// Operation Mode
// bOutputManAuto := GVL_IO.aOutputCmd[1].11; //Temp Controller Mode Command
// nOutputManAutoBytes.0 	:= GVL_IO.aOutputCmd[1].11; //Command

IF nInputManAutoBytes.0 THEN // Read form E3508 Mode, 1:Man 0:Auto
	wOutputPowerSVBytes 	:= WORD_TO_USINT_Bit(wControlValue*10); //multiple to 10, Power Reate Set Value
	aOutputPowerBytes[1] 	:= wOutputPowerSVBytes.Lower;
	aOutputPowerBytes[2] 	:= wOutputPowerSVBytes.Upper;
ELSE
	wOutputSVBytes 			:= WORD_TO_USINT_Bit(wControlValue); // Temperature Set Value
	aOutputSVBytes[1] 		:= wOutputSVBytes.Lower;
	aOutputSVBytes[2] 		:= wOutputSVBytes.Upper;
END_IF

(* Write to Induction Heater Value *)
GVL_IO.aDigitalOutputIO[2].0 := bHeaterOn;
GVL_IO.aDigitalOutputIO[2].1 := bHeaterReset;
GVL_IO.nE3508_nInputManAutoBytes := nInputManAutoBytes; //State

END_PROGRAM

// ---- FUNTION/USINT_TO_WORD_Bit.TcPOU
//2-USINT combine to 1-WORD converting using a bit operation
FUNCTION USINT_TO_WORD_Bit : WORD
VAR_INPUT
	aInput_L : USINT; //Lower
	aInput_U : USINT; //Upper
END_VAR
VAR
	nWord_L : WORD; //Lower
	nWord_U : WORD; //Upper
END_VAR

nWord_L := TO_WORD(aInput_L);
// 1111_1111
// 0000_0000_1111_1111
nWord_U := TO_WORD(aInput_U);
// 1111_1111
// 0000_0000_1111_1111
nWord_U := SHL(nWord_U, 8);
// 1111_1111_0000_0000
USINT_TO_WORD_Bit := TO_WORD(nWord_L OR nWord_U);

END_FUNCTION

// ---- FUNTION/WORD_TO_USINT_Bit.TcPOU
// 1-WORD divide to 2-USINT
FUNCTION WORD_TO_USINT_Bit : outWord
VAR_INPUT
	nOutput : WORD;
END_VAR
VAR
	outWord : outWord;
END_VAR

outWord.Lower := TO_USINT(nOutput); //Lower Bits
outWord.Upper := TO_USINT(SHR(nOutput, 8)); //Uppper Bits
WORD_TO_USINT_Bit := outWord;

END_FUNCTION

// ---- POUs/P12_IQ_PLUS.TcPOU
PROGRAM P12_IQ_PLUS
VAR
	wControlValue 		: WORD := 760;//Pressure Set Value
	wCDG1_PV 			: WORD; //CD2 Current Pressure
	wCDG2_PV 			: WORD; //CD2 Current Pressure
	bVacuumPumpCB		: BOOL;
	bThrottleValveCP	: BOOL;

	//nInputStatus
	ingPressureControl 		: BOOL;
	ingPositionControl 		: BOOL;
	isValveOpen 			: BOOL;
	isValveNotInitialized 	: BOOL;	
	isValveClosed 			: BOOL;
	isValveFaultState 		: BOOL;
	ingValveInitializing 	: BOOL;
	ingHoldState 			: BOOL;
	
	// Vacuum Pump Status
	isPumpFault				: BOOL;
	isPumpWarning			: BOOL;
	isPumpAlarm				: BOOL;
	isFBRunning				: BOOL;
// 	isPumpRunning			: BOOL;
	//wSetPoint 			: WORD; //Set Point
	nTValveMode 		: USINT := 0; //Valve Mode
	bPumpOn				: BOOL;
	bPumpReset			: BOOL;	//Input from IQ-PLUS Throttle Valve
	
	nInputStatus AT %I* : USINT; //Input Status Bytes
	aInputPressurePV_CDG1 AT %I* : ARRAY[1..2]OF USINT; //CDG1 Pressure
	aInputPressurePV_CDG2 AT %I* : ARRAY[1..2]OF USINT; //CDG2 Pressure
	aInputPressureSP AT %I* : ARRAY[1..2]OF USINT; //Set Point Pressure
	aInputValvePosionPV AT %I* : ARRAY[1..2]OF USINT; //Current Valve Position
	
	wTypedControlValue 	: WORD;
	wOutputSVBytes : outWord; //Word to Byte variable
	nSetType 			: USINT; //1:Pressure Conrol, 2:Position Control
	
	//Output to IQ-PLUS Throttle Valve
	nOutputMode AT %Q* : USINT;
	aOutputSVBytes AT %Q* : ARRAY[1..2]OF USINT; //Set Pressure
	nOutputSetType AT %Q* : USINT; //1:Pressure Control, 2:Valve Position Control

	wByteCDG1_PV 			: WORD; //CDG1 Current Pressure, Not Used
	wByteCDG2_PV 			: WORD; //CDG2 Current Pressure
	wByteValvePosition_PV : WORD; //Current Valve Position (0~100%)
	nInputStatusOld : USINT := 9; //Value Change Monitoring, First Temp value
END_VAR

VAR CONSTANT
	//Conversion Parameter
	SetPointFactor : REAL := 327.67; //Range 0~7FFFh
	PressureFactor : REAL := 24.576;	//Range 0~6000h
END_VAR

//Model : IQ Plus 
//Pressure Range : 0 ~ 1,000 Torr
IF GVL_IO.aOutputCmd[1].12 THEN // Pressure Mode Setting
	nOutputSetType := 1; // Pressure Control
ELSE
	nOutputSetType := 2; // Position Control
END_IF

(* Command *)
bPumpOn 			:= GVL_IO.aOutputCmd[1].6;
bPumpReset 			:= GVL_IO.aOutputCmd[1].7;

(* Read from Power Distribution Pannel *)
bVacuumPumpCB		:= GVL_IO.aDigitalInputIO[5].1;
bThrottleValveCP 	:= GVL_IO.aDigitalInputIO[5].5; //Throttle Valve CP

(* Read from Vacuum Pump *)
isPumpFault			:= GVL_IO.aDigitalInputIO[2].7;
isPumpWarning		:= GVL_IO.aDigitalInputIO[3].0;
isPumpAlarm			:= GVL_IO.aDigitalInputIO[3].1;
isFBRunning			:= GVL_IO.aDigitalInputIO[3].2;
// isPumpRunning		:= GVL_IO.aDigitalInputIO[3].3;

(* Read from Device Value *)
// 2USINT to WORD
wByteCDG1_PV 		:= USINT_TO_WORD_Bit(aInputPressurePV_CDG1[1],aInputPressurePV_CDG1[2]);
wByteCDG2_PV 		:= USINT_TO_WORD_Bit(aInputPressurePV_CDG2[1],aInputPressurePV_CDG2[2]);
wByteValvePosition_PV 	:= USINT_TO_WORD_Bit(aInputValvePosionPV[1], aInputValvePosionPV[2]);
wControlValue		:= LREAL_TO_WORD(GVL_IO.aController[28].rControlValue);

//From IQ Plus
// wCDG1_PV 			:= REAL_TO_WORD(wByteCDG1_PV/PressureFactor);
// wCDG2_PV 			:= REAL_TO_WORD(wByteCDG2_PV/PressureFactor);
GVL_IO.wIqPlus_CDG1_PV 	:= REAL_TO_WORD(wByteCDG1_PV/PressureFactor);
GVL_IO.wIqPlus_CDG2_PV 	:= REAL_TO_WORD(wByteCDG2_PV/PressureFactor);

//To IQ Plus
nOutputMode := WORD_TO_USINT(GVL_IO.aOutputCmd[2]); //Throttle Valve Mode Setting 0:Normal 1:Close 2:Open 3:Hold 4:Reset
IF nOutputMode = 0 AND nSetType = 1 THEN
	wTypedControlValue := REAL_TO_WORD(wControlValue * SetPointFactor * 0.1); //Pressure Control
ELSIF nOutputMode = 0 AND nSetType = 2 THEN
	wTypedControlValue := REAL_TO_WORD(wControlValue * SetPointFactor); // Position Control
END_IF

wOutputSVBytes 		:= WORD_TO_USINT_Bit(wTypedControlValue);
aOutputSVBytes[1] 	:= wOutputSVBytes.Lower;
aOutputSVBytes[2] 	:= wOutputSVBytes.Upper;

//Valve Status Initailize
IF nInputStatus <> nInputStatusOld THEN
	// Staus Initializing
	ingPressureControl := FALSE;
	ingPositionControl := FALSE;
	isValveOpen := FALSE;
	isValveNotInitialized := FALSE;	
	isValveClosed := FALSE;
	isValveFaultState := FALSE;
	ingValveInitializing := FALSE;
	ingHoldState := FALSE;
	// Status Update	
	nInputStatusOld := nInputStatus;
END_IF

//Update Valve Status
CASE nInputStatus OF
	0 : ingPressureControl := TRUE; //Pressure Control Performing.
	1 : ingPositionControl := TRUE; //Position Control Performing.	
	2 : isValveOpen := TRUE; //Valve Open, Stopped, Not Controlling.
	3 : isValveNotInitialized := TRUE; //Valve not initialized power on or RESET Command.
	4 : isValveClosed := TRUE; //Valve Closed, Stopped, Not Controlling.
	5 : isValveFaultState := TRUE; //Has faulted during valve initialization or operation.
	6 : ingValveInitializing := TRUE; //Initailizing Process.
	8 : ingHoldState := TRUE; //intermediate position, not at open or close and not controlling pressure.
END_CASE

// nOutputMode
// 0 : uses setpoint and setpoint type to control the valve.
// 1 : Does not use setpoint and setpoint type to operate the valve.
// 2 : Does not use setpoint and setpoint type to operate the valve.
// 3 : Holds valve in current position.
// 4 : Reset the controller.

GVL_IO.nIQPLUS_SetType 	:= nOutputSetType;
GVL_IO.nIQPLUS_Mode 	:= nOutputMode;

GVL_IO.aMonitoring_PV[11] := wByteValvePosition_PV/SetPointFactor;
GVL_IO.aDigitalOutputIO[2].2 := bPumpOn; //Pump On
GVL_IO.aDigitalOutputIO[2].3 := bPumpReset; // Pump Reset
GVL_IO.isPumpRunning := GVL_IO.aDigitalInputIO[3].3;

END_PROGRAM

// ---- POUs/P13_LineHeater.TcPOU
PROGRAM P13_LineHeater
VAR
	rTemperatureSV 		: ARRAY[1..8]OF REAL;
	bAutoTuneSV 		: ARRAY[1..8]OF BOOL;

	rTemperaturePV 		: ARRAY[1..8]OF REAL;
	isLineHeater_Run	: ARRAY[1..8]OF BOOL;
	isLineHeater_ATune	: ARRAY[1..8]OF BOOL;
	isLineHeater_Err	: ARRAY[1..8]OF BOOL;

	TimeOnDelay			: TON; //Time delay after Power ON of Thermal Bath
	TimeCycle			: TON;
	nComMode 			: INT; // //1 = PV Req, 2 = STATUS Req, 3 = SV Write, 4 = AutoTune On/Off
	nCount 				: INT;
	rTemperatureTV 		: ARRAY[1..8]OF REAL;
	bAutoTuneTV			: ARRAY[1..8]OF BOOL;

	//for sending variable
	TimeWaitSend		:TON;
	bSendingEnable 		: BOOL:=TRUE; // Check the Sending Stage
	bSetValueMode 		: BOOL;
	fbSend				: SendString;
	sSendString 		: STRING;
	bSendBusy			: BOOL;
	bSendingOK 			: BOOL; //v1
	eSendErrorID		: ComError_t;
	
	// for received variable
	TimeWaitReceive		:TON;
	fbReceive			: ReceiveString;
	sReceivedString		: STRING;
	bStringReceived		: BOOL;
	bReceiveBusy		: BOOL;
	bReceiveError		: BOOL;
	eReceiveErrorID		: ComError_t;
	bReceiveTimeout		: BOOL;
	bReceivedOK 		: BOOL;
	hStrReceivedST		: STRING;
	hStrReceivedPV		: STRING;
	
	nHeaterNumber 		: INT := 1;
	sHeaterNumber 		: STRING := '1';
	sReceivedHeaterNumber : STRING;
	nReceivedHeaterNumber : INT;
	sReceivedAffirmation : STRING;
	sReceivedData 		: STRING;
	nHeaterStrPositionPV : INT:= 11; //Received String Start Position
	nDecimal			:INT;
	nSendStrCounter		:INT := 1;
	bReset : BOOL;
	sTest : STRING;
	nStrPosition : INT;
	nHeaterNumberPV : INT;
	sTemperaturePV : STRING;
	(* Input *)
	bLineHeaterCB		: BOOL;
	bLineHeaterCP		: BYTE;
END_VAR

//LH: Line Heater x 8EA -> 8Channel TIC 1EA
//Maker: HANYOUNG NUX
//Model: MC9-8RD0SS32
//Temp Range: -15 ~200℃
//RS485: 9600, DataBit(8), Parity(None), StopBit(1)
//BCC Check X

(* Read from Device Value *)
// Line Heater CP
bLineHeaterCB	:= GVL_IO.aDigitalInputIO[5].2;
bLineHeaterCP 	:= GVL_IO.aDigitalInputIO[6]; //LineHeaterCP1   := bLineHeaterCP.0, Until CP8

// make a sending string
TimeOnDelay(IN:= P90_Interlock.bLineHeaterMC, PT :=T#5S); //Time Delay after a Thermal Bath MC ON
IF TimeOnDelay.Q THEN
	TimeOnDelay(IN:=FALSE);
	// Make a sending string Set value or Request value 
	IF bSendingEnable = FALSE THEN
		bSendingEnable := TRUE;
		bSendingOK := FALSE;
		bReceivedOK := FALSE;
		
		IF nComMode <>1 THEN
			sSendString := '$0201DRS,08,0001$0D$0A'; //Request PV
			nComMode := 1;
		ELSE
			sSendString := '$0201DRS,08,0111$0D$0A'; //Request State
			nComMode := 2;
		END_IF
	
		FOR nHeaterNumber:= 1 TO 8 DO
			IF (rTemperatureTV[nHeaterNumber] <> rTemperatureSV[nHeaterNumber]) THEN
				// if SetValue are different to TargetValue, change Target vale to setvalue
				rTemperatureTV[nHeaterNumber] := rTemperatureSV[nHeaterNumber];
				sSendString := Real_To_String_LineHeater(rTemperatureTV[nHeaterNumber]*10, nHeaterNumber); //Move the decimal point by 1
			END_IF
			IF (bAutoTuneSV[nHeaterNumber] <> bAutoTuneTV[nHeaterNumber]) THEN
				bAutoTuneTV[nHeaterNumber] := bAutoTuneSV[nHeaterNumber];
				sSendString := BOOL_TO_STRING_LHeaterON(nHeaterNumber,bAutoTuneTV[nHeaterNumber]);
			END_IF
			
				TimeWaitSend(IN:=TRUE, PT:=T#10MS);
				IF TimeWaitSend.Q THEN
					TimeWaitSend(IN:=FALSE);
					IF fbSend.Busy THEN
						fbSend(	SendString:= sSendString,
							TXbuffer:= TxBufferLH,
							Busy=> bSendBusy,
							Error=> );
						IF fbSend.Error <> COMERROR_NOERROR THEN
							eSendErrorID := fbSend.Error;
							bSendingOK := FALSE;
						ELSE
							eSendErrorID := COMERROR_NOERROR;
							bSendingOK := TRUE;
						END_IF
					END_IF
				END_IF

		END_FOR
		
	END_IF
	
	TimeWaitSend(IN:=bSendingEnable AND bSendingOK = FALSE, PT:=T#10MS);
	IF TimeWaitSend.Q OR fbSend.Busy THEN
		bSendingOK := TRUE;
		fbSend(
			SendString := sSendString,
			TXBuffer := TXBufferLH,
			Busy => bSendBusy,
			Error =>
			);
		IF fbSend.Error <> COMERROR_NOERROR THEN
			eSendErrorID := fbSend.Error;
			bSendingOK := FALSE;
		ELSE
			bSendingOK := TRUE;
			bSendingOK := TRUE;
		END_IF
	END_IF
	
	fbReceive(
		Prefix := '$02',
		Suffix:= '$0D$0A',
		Timeout:= T#1S,
		ReceivedString:= sReceivedString,
		RXbuffer:=RXbufferLH,
		StringReceived=> bStringReceived,
		Busy=> bReceiveBusy,
		Error=>
		);
	IF bStringReceived THEN
		bStringReceived := FALSE;
		bReceivedOK:= TRUE;
		
		IF nComMode =1 THEN
			nStrPosition := 11;			
			FOR nHeaterNumber := 1 TO 8 DO
				hStrReceivedPV := MID(STR:=sReceivedString, LEN:=4, POS:=nStrPosition);
				rTemperaturePV[nHeaterNumber] := (HEXSTR_TO_REAL_LHeaterPV(hStrReceivedPV))/10; //Move the decimal point by 1
				nStrPosition := nStrPosition + 5;
			END_FOR
		ELSE
			nStrPosition := 11;		
			FOR nHeaterNumber := 1 TO 8 DO
				hStrReceivedST := MID(STR:=sReceivedString, LEN:=4, POS:=nStrPosition);						
				IF hStrReceivedST = '0002' THEN
					isLineHeater_Run[nHeaterNumber] 	:= TRUE;
					isLineHeater_ATune[nHeaterNumber] 	:= FALSE;
					isLineHeater_Err[nHeaterNumber] 	:= FALSE;
				ELSIF hStrReceivedST = '0004' THEN
					isLineHeater_Run[nHeaterNumber] 	:= FALSE;
					isLineHeater_ATune[nHeaterNumber] 	:= TRUE;
					isLineHeater_Err[nHeaterNumber] 	:= FALSE;
				ELSIF hStrReceivedST = '0080' THEN
					isLineHeater_Run[nHeaterNumber] 	:= FALSE;
					isLineHeater_ATune[nHeaterNumber] 	:= FALSE;
					isLineHeater_Err[nHeaterNumber] 	:= TRUE;
				ELSE
					isLineHeater_Run[nHeaterNumber] 	:= FALSE;
					isLineHeater_ATune[nHeaterNumber] 	:= FALSE;
					isLineHeater_Err[nHeaterNumber] 	:= FALSE;
				END_IF
				nStrPosition := nStrPosition + 5;		
			END_FOR
		END_IF
	END_IF
	
	TimeWaitReceive(IN:=bReceivedOK,PT:=T#1S);
	TimeCycle(IN:=TRUE, PT:=T#2S);
	IF TimeWaitReceive.Q OR TimeCycle.Q THEN
		TimeWaitReceive(IN:= TRUE);
		TimeCycle(IN:= FALSE);
		bSendingEnable := FALSE;
	END_IF
END_IF
GVL_IO.aLineHeater_rTemperaturePV := rTemperaturePV;

END_PROGRAM

// ---- POUs/P90_Interlock.TcPOU
PROGRAM P90_Interlock
VAR
	bRecipeRunning 		: BOOL;
	RecipeStopped 		: BOOL;
	ManualOperation 	: BOOL;
	bInductionHeaterMC	: BOOL;
	bThermalBathMC		: BOOL;
	bVacuumPumpMC 		: BOOL;
	bLineHeaterMC 		: BOOL; 

	bRecipeStartAvailable	: BOOL;
	bReactorOpenEnable		: BOOL;
	bHeaterOnEnable			: BOOL;
	bPumpOnEnable			: BOOL;
	
	bDorOnEnable			: BOOL;
	bDorOffEnable			: BOOL;
	bOpenEnableTemp			: BOOL;
	bOpenEnablePress		: BOOL;	
	
	bPowerResetSwitch		: BOOL;
	bMainPowerMonitor		: BOOL;

	AlarmTrig				: BOOL;
	WarningTrig				: BOOL;
	bMaintKey				: BOOL;
	bGasStateProcess		: BOOL;
	bGasStateSource			: BOOL;
	bGasStateVent			: BOOL;

	bPowerResetLED			: BOOL;
	bUPSMode				: BOOL;
	tAlarmDelay_A			: TIME; //아날로그 디바이스 지연시간
	tAlarmDelay_D			: TIME; //디지털 디바이스 지연시간
	
	fbDeviationCheck		:ARRAY[1..29] OF FB_DeviationCheck;
	wDeviceAlarmEnable		: DWORD;
	wDeviceWarningEnable	: DWORD;
	bDeviationAlarm			: BOOL;
	bDeviationWarning		: BOOL;
	wDeviationAlarm			: DWORD;
	wDeviationWarning		: DWORD;

	fbSensorLimitCheck		:ARRAY[1..4] OF FB_SensorLimitCheck;
	wLimitAlarmEnable		: DWORD;
	wLimitWarningEnable		: DWORD;
	bLimitAlarm				: BOOL;
	bLimitWarning			: BOOL;
	wLimitAlarm				: DWORD;
	wLimitWarning			: DWORD;
	
	fbFaultCheck			:ARRAY[1..8] OF FB_FaultCheck;
	wAlarmEnable			: DWORD;
	wWarningEnable			: DWORD;

	bFaultAlarm				: BOOL;
	bFaultWarning			: BOOL;
	wAlarm					: DWORD;
	wWarning				: DWORD;
		
	bAlarmEnable			: BOOL;
	bWarningEnable			: BOOL;
	bDeviceCurrentAlarmState	: BOOL;
	bDeviceCurrentWarningState 	: BOOL;
	fDeviceCurrentValue			: REAL;
	fDeviceAlarmTreshold		: REAL;
	fDeviceWarningTreshold		: REAL;
	
	i	: INT;
	j 	: INT;

END_VAR

(* Read from Device*)
//Interlock Variable Set
bMaintKey := GVL_IO.aDigitalInputIO[1].0;
bPowerResetSwitch := GVL_IO.aDigitalInputIO[1].1;
bMainPowerMonitor := GVL_IO.aDigitalInputIO[7].5;
bGasStateProcess := NOT(GVL_IO.aOutputSolValve[1].0) AND //HYD Carrier Change Valve
	NOT(GVL_IO.aOutputSolValve[1].1) AND //Main Carrier Change Valve
	NOT(GVL_IO.aOutputSolValve[1].2) AND //SiH4 Source Change Valve
	NOT(GVL_IO.aOutputSolValve[1].3) //NH3 Source Change Valve
	; //All False이면 Safety State
bGasStateSource := NOT(GVL_IO.aOutputSolValve[1].4) AND NOT(GVL_IO.aOutputSolValve[1].5) AND NOT(GVL_IO.aOutputSolValve[1].6) AND //Source #1
	NOT(GVL_IO.aOutputSolValve[1].7) AND NOT(GVL_IO.aOutputSolValve[1].8) AND NOT(GVL_IO.aOutputSolValve[1].9) AND //Source #2
	NOT(GVL_IO.aOutputSolValve[1].10) AND NOT(GVL_IO.aOutputSolValve[1].11) AND NOT(GVL_IO.aOutputSolValve[1].12) AND //Source #3
	NOT(GVL_IO.aOutputSolValve[1].13) AND NOT(GVL_IO.aOutputSolValve[1].14) AND NOT(GVL_IO.aOutputSolValve[1].15) AND //Source #4
	NOT(GVL_IO.aOutputSolValve[2].0) AND NOT(GVL_IO.aOutputSolValve[2].1) AND NOT(GVL_IO.aOutputSolValve[2].2) AND //Source #5
	NOT(GVL_IO.aOutputSolValve[2].3) AND NOT(GVL_IO.aOutputSolValve[2].4) AND NOT(GVL_IO.aOutputSolValve[2].6) //Source #6
	; //All False이면 Safety State
bGasStateVent := NOT(GVL_IO.aOutputSolValve[2].15);
GVL_IO.aInterlock[1].10 := bRecipeStartAvailable;
GVL_IO.aInterlock[1].11 := bReactorOpenEnable;
GVL_IO.aInterlock[1].12 := bHeaterOnEnable;
GVL_IO.aInterlock[1].13 := bPumpOnEnable;

//알람 지연 시간 변환
tAlarmDelay_A := REAL_TO_TIME(GVL_IO.aInterlockSet[3]*1000); // UI Setting Analog Delay Time Value(Miliseconde)
tAlarmDelay_D := REAL_TO_TIME(GVL_IO.aInterlockSet[4]*1000);

//Sinal Tower Set
//Controller Deviation Monitoring - MFC/EPC
IF bMaintKey THEN //bMaintKey 변경
	//매인터넌스 키가 ON 되었을 때 MC(Induction, Bath, Pump, L_Heater) 조작 허용
	GVL_IO.nCaseSignalTower	:= 4; //Signal Tower Blue - Maintenance
	GVL_IO.aDigitalOutputIO[3].0 := GVL_IO.aOutputCmd[1].0;
	GVL_IO.aDigitalOutputIO[3].1 := GVL_IO.aOutputCmd[1].1;
	GVL_IO.aDigitalOutputIO[3].2 := GVL_IO.aOutputCmd[1].2;
	GVL_IO.aDigitalOutputIO[3].3 := GVL_IO.aOutputCmd[1].3;
ELSE
	FOR i := 1 TO 26 DO
		wDeviceAlarmEnable := SHR(GVL_IO.aInterlockEnable[2], (i+2)); //오늘쪽 쉬프트 연산
		wDeviceWarningEnable := SHR(GVL_IO.aInterlockEnable[3], (i+2));
		fbDeviationCheck[i](
			bAlarmEnable := wDeviceAlarmEnable.0,
			bWarningEnable := wDeviceWarningEnable.0,
			fCurrentValue := GVL_IO.aController_PV[i],
			fControlValue := LREAL_TO_REAL(GVL_IO.aController[i].rControlValue),
			fMaxValue := GVL_IO.AnalogControllerOutputVoltage,
			fAlarmTreshold := GVL_IO.aInterlockSet[1],
			fWarningTreshold := GVL_IO.aInterlockSet[2],
			tAlarmDelay := tAlarmDelay_A,
			bDeviationAlarm => bDeviationAlarm, //알람 출력
			bDeviationWarning => bDeviationWarning // 주의(Warning) 출력
			);
		IF bDeviationAlarm THEN
			GVL_IO.aInterlock[1].0 := TRUE; //Alarm Trig
			GVL_IO.nCaseSignalTower := 1; // Signal Tower RED - Alarm
			wDeviationAlarm := ROR(GVL_IO.aInterlock[3], (i+2));
			wDeviationAlarm.0 := TRUE;
			GVL_IO.aInterlock[3] := ROL(wDeviationAlarm, (i+2));
		ELSE
			wDeviationAlarm := ROR(GVL_IO.aInterlock[3], (i+2));
			wDeviationAlarm.0 := FALSE;
			GVL_IO.aInterlock[3] := ROL(wDeviationAlarm, (i+2));	
		END_IF
		
		IF bDeviationWarning THEN
			GVL_IO.aInterlock[1].1 := TRUE; // Warning Trig
			GVL_IO.nCaseSignalTower := 2; // Signal Tower Yellow - Warning
			wDeviationWarning := ROR(GVL_IO.aInterlock[5], (i+2));
			wDeviationWarning.0 := TRUE;
			GVL_IO.aInterlock[5] := ROL(wDeviationWarning, (i+2));
		ELSE
			wDeviationWarning := ROR(GVL_IO.aInterlock[5], (i+2));
			wDeviationWarning.0 := FALSE;
			GVL_IO.aInterlock[5] := ROL(wDeviationWarning, (i+2));
		END_IF
	END_FOR
	//Controller Deviation Monitoring - Temp, Pressure, Rotation
	FOR i := 27 TO 29 DO
		wDeviceAlarmEnable := SHR(GVL_IO.aInterlockEnable[2], (i-27)); //오늘쪽 쉬프트 연산, -27은 어레이 변수 옵셋값
		wDeviceWarningEnable := SHR(GVL_IO.aInterlockEnable[3], (i-27));
		fbDeviationCheck[i](
			bAlarmEnable := wDeviceAlarmEnable.0,
			bWarningEnable := wDeviceWarningEnable.0,
			fCurrentValue := GVL_IO.aController_PV[i],
			fControlValue := LREAL_TO_REAL(GVL_IO.aController[i].rControlValue),
			fMaxValue := GVL_IO.aReactorMaxValue[i - 26],
			fAlarmTreshold := GVL_IO.aInterlockSet[1],
			fWarningTreshold := GVL_IO.aInterlockSet[2],
			tAlarmDelay := tAlarmDelay_A,
			bDeviationAlarm => bDeviationAlarm, //알람 출력
			bDeviationWarning => bDeviationWarning // 주의(Warning) 출력
			);
		IF bDeviationAlarm THEN
			GVL_IO.aInterlock[1].0 := TRUE; //Alarm Trig
			GVL_IO.nCaseSignalTower := 1; // Signal Tower RED - Alarm
			wDeviationAlarm := ROR(GVL_IO.aInterlock[3], (i-27));
			wDeviationAlarm.0 := TRUE;
			GVL_IO.aInterlock[3] := ROL(wDeviationAlarm, (i-27));
		ELSE
			wDeviationAlarm := ROR(GVL_IO.aInterlock[3], (i-27));
			wDeviationAlarm.0 := FALSE;
			GVL_IO.aInterlock[3] := ROL(wDeviationAlarm, (i-27));
		END_IF
		IF bDeviationWarning THEN
			GVL_IO.aInterlock[1].1 := TRUE; // Warning Trig
			GVL_IO.nCaseSignalTower := 2; // Signal Tower Yellow - Warning
			wDeviationWarning := ROR(GVL_IO.aInterlock[5], (i-27));
			wDeviationWarning.0 := TRUE;
			GVL_IO.aInterlock[5] := ROL(wDeviationWarning, (i-27));
		ELSE
			wDeviationWarning := ROR(GVL_IO.aInterlock[5], (i-27));
			wDeviationWarning.0 := FALSE;
			GVL_IO.aInterlock[5] := ROL(wDeviationWarning, (i-27));
		END_IF	
	END_FOR
	//Gas Pressure Alarm N2, H2, NH3, SiH4
	FOR i := 1 TO 4 DO
		wLimitAlarmEnable := SHR(GVL_IO.aInterlockEnable[4], (i-1)); //오늘쪽 쉬프트 연산, 은 어레이 변수 옵셋값
		wLimitWarningEnable := SHR(GVL_IO.aInterlockEnable[5], (i-1));
		fbSensorLimitCheck[i](
			bAlarmEnable := wLimitAlarmEnable.0,
			bWarningEnable := wLimitWarningEnable.0,
			fCurrentValue := GVL_IO.aMonitoring_PV[(i+3)],
			fAlarmTreshold := GVL_IO.aInterlockSet[5],
			fWarningTreshold := GVL_IO.aInterlockSet[6],
			tAlarmDelay := tAlarmDelay_D,
			bLimitAlarm => bLimitAlarm, //알람 출력
			bLimitWarning => bLimitWarning //주의(Warning) 출력
			);	
		IF bLimitAlarm THEN		
			GVL_IO.aInterlock[1].0 := TRUE; //Alarm Trig
			GVL_IO.nCaseSignalTower := 1; // Signal Tower RED - Alarm
			//팝업 표시
			wLimitAlarm := ROR(GVL_IO.aInterlock[2], (i-1));
			wLimitAlarm.0 := TRUE;
			GVL_IO.aInterlock[2] := ROL(wLimitAlarm, (i-1));
			//대시보드 표시
			wLimitAlarm := ROR(GVL_IO.aInterlock[1], (i*2));
			wLimitAlarm.0 := TRUE;
			GVL_IO.aInterlock[1] := ROL(wLimitAlarm, (i*2));
		ELSE
			//팝업 표시
			wLimitAlarm := ROR(GVL_IO.aInterlock[2], (i-1));
			wLimitAlarm.0 := FALSE;
			GVL_IO.aInterlock[2] := ROL(wLimitAlarm, (i-1));
			//대시보드 표시
			wLimitAlarm := ROR(GVL_IO.aInterlock[1], (i*2));
			wLimitAlarm.0 := FALSE;
			GVL_IO.aInterlock[1] := ROL(wLimitAlarm, (i*2));
		END_IF
		
		IF bLimitWarning THEN		
			GVL_IO.aInterlock[1].1 := TRUE; //Warning Trig
			GVL_IO.nCaseSignalTower := 2; // Signal Tower YELLOW - Warning
			//팝업 표시
			wLimitWarning := ROR(GVL_IO.aInterlock[4], (i-1));
			wLimitWarning.0 := TRUE;
			GVL_IO.aInterlock[4] := ROL(wLimitWarning, (i-1));
			//대시보드 표시
			wLimitWarning := ROR(GVL_IO.aInterlock[1], (i*2)+1);
			wLimitWarning.0 := TRUE;
			GVL_IO.aInterlock[1] := ROL(wLimitWarning, (i*2)+1);
		ELSE
			//팝업 표시
			wLimitWarning := ROR(GVL_IO.aInterlock[4], (i-1));
			wLimitWarning.0 := FALSE;
			GVL_IO.aInterlock[4] := ROL(wLimitWarning, (i-1));
			//대시보드 표시
			wLimitWarning := ROR(GVL_IO.aInterlock[1], (i*2)+1);
			wLimitWarning.0 := FALSE;
			GVL_IO.aInterlock[1] := ROL(wLimitWarning, (i*2)+1);
		END_IF
	END_FOR
	
	//Cooling Water Over Temperature, Susceptor Over Temperature, Reactor Over Pressure
	FOR i := 1 TO 4 DO
		CASE i OF
			1: //CW Temperature High S/H
				bAlarmEnable := GVL_IO.aInterlockEnable[4].4;
				bWarningEnable := GVL_IO.aInterlockEnable[5].4;
				fDeviceCurrentValue := GVL_IO.aMonitoring_PV[8];
				fDeviceAlarmTreshold := GVL_IO.aInterlockSet[7];
				fDeviceWarningTreshold := GVL_IO.aInterlockSet[8];
			2: //CW Temperature High Coil
				bAlarmEnable := GVL_IO.aInterlockEnable[4].5;
				bWarningEnable := GVL_IO.aInterlockEnable[5].5;
				fDeviceCurrentValue := GVL_IO.aMonitoring_PV[9];
				fDeviceAlarmTreshold := GVL_IO.aInterlockSet[9];
				fDeviceWarningTreshold := GVL_IO.aInterlockSet[10];
			3: //Susceptor Over Temperature
				bAlarmEnable := GVL_IO.aInterlockEnable[4].6;
				bWarningEnable := GVL_IO.aInterlockEnable[5].6;
				fDeviceCurrentValue := GVL_IO.aController_PV[27];
				fDeviceAlarmTreshold := GVL_IO.aInterlockSet[11];
				fDeviceWarningTreshold := (GVL_IO.aInterlockSet[11] - 20.0); //20도 아래에서 Warning 발생				
			4: //Reactor Over Pressure Alarm
				bAlarmEnable := GVL_IO.aInterlockEnable[4].7;
				bWarningEnable := GVL_IO.aInterlockEnable[5].7;
				fDeviceCurrentValue := GVL_IO.aController_PV[28];
				fDeviceAlarmTreshold := GVL_IO.aInterlockSet[12];
				fDeviceWarningTreshold := (GVL_IO.aInterlockSet[12] - 50.0); //50Torr 아래에서 Warning 발생							
		END_CASE
		fbSensorLimitCheck[i](
			bAlarmEnable := bAlarmEnable,
			bWarningEnable := bWarningEnable,
			fCurrentValue := fDeviceCurrentValue,
			fAlarmTreshold := fDeviceAlarmTreshold,
			fWarningTreshold := fDeviceWarningTreshold,
			tAlarmDelay := tAlarmDelay_D,
			bLimitAlarm => bLimitAlarm, //알람 출력
			bLimitWarning => bLimitWarning //주의(Warning) 출력
			);
		IF bLimitAlarm THEN		
			GVL_IO.aInterlock[1].0 := TRUE; //Alarm Trig
			GVL_IO.nCaseSignalTower := 1; // Signal Tower RED - Alarm
			wDeviationAlarm := ROR(GVL_IO.aInterlock[2], (i+3));
			wDeviationAlarm.0 := TRUE;
			GVL_IO.aInterlock[2] := ROL(wDeviationAlarm, (i+3));
		ELSE
			wDeviationAlarm := ROR(GVL_IO.aInterlock[2], (i+3));
			wDeviationAlarm.0 := FALSE;
			GVL_IO.aInterlock[2] := ROL(wDeviationAlarm, (i+3));
		END_IF
		
		IF bDeviationWarning THEN
			GVL_IO.aInterlock[1].1 := TRUE; // Warning Trig
			GVL_IO.nCaseSignalTower := 2; // Signal Tower Yellow - Warning
			wDeviationWarning := ROR(GVL_IO.aInterlock[4], (i+3));
			wDeviationWarning.0 := TRUE;
			GVL_IO.aInterlock[4] := ROL(wDeviationWarning, (i+3));
		ELSE
			wDeviationWarning := ROR(GVL_IO.aInterlock[4], (i+3));
			wDeviationWarning.0 := FALSE;
			GVL_IO.aInterlock[4] := ROL(wDeviationWarning, (i+3));
		END_IF		
	END_FOR
	
	//Device Fault Check - Pneumatic, Heater, Pump, Motor, GC Door, RC Door
	FOR i := 1 TO 8 DO
		CASE i OF
			1: //CDA Alarm Switch (Pneumatic)
				bAlarmEnable := GVL_IO.aInterlockEnable[4].8;
				bWarningEnable := GVL_IO.aInterlockEnable[5].8;
				bDeviceCurrentAlarmState := GVL_IO.aInputState[1].4;
				bDeviceCurrentWarningState := GVL_IO.aInputState[1].4;
			2: //Cooling Water Switch
				bAlarmEnable := GVL_IO.aInterlockEnable[4].9;
				bWarningEnable := GVL_IO.aInterlockEnable[5].9;
				bDeviceCurrentAlarmState := GVL_IO.aInputState[1].5;
				bDeviceCurrentWarningState := GVL_IO.aInputState[1].5;
			3: //Induction Heater Fault
				bAlarmEnable := GVL_IO.aInterlockEnable[4].10;
				bWarningEnable := GVL_IO.aInterlockEnable[5].10;
				bDeviceCurrentAlarmState := GVL_IO.aInputState[1].8;
				bDeviceCurrentWarningState := GVL_IO.aInputState[1].8;
			4: //Rotatin Motor Fault
				bAlarmEnable := GVL_IO.aInterlockEnable[4].11;
				bWarningEnable := GVL_IO.aInterlockEnable[5].11;
				bDeviceCurrentAlarmState := GVL_IO.aInputState[1].11;
				bDeviceCurrentWarningState := GVL_IO.aInputState[1].11;
			5: //Vacuum Pump Fault
				bAlarmEnable := GVL_IO.aInterlockEnable[4].12;
				bWarningEnable := GVL_IO.aInterlockEnable[5].12;
				bDeviceCurrentAlarmState := GVL_IO.aInputState[1].12;
				bDeviceCurrentWarningState := GVL_IO.aInputState[1].14;
			6: //Gas Cabinet Door Open
				bAlarmEnable := GVL_IO.aInterlockEnable[4].13;
				bWarningEnable := GVL_IO.aInterlockEnable[5].13;
				bDeviceCurrentAlarmState := GVL_IO.aInputState[2].0;
				bDeviceCurrentWarningState := GVL_IO.aInputState[2].0;
			7: //Reactor Cabinet Door Open
				bAlarmEnable := GVL_IO.aInterlockEnable[4].14;
				bWarningEnable := GVL_IO.aInterlockEnable[5].14;
				bDeviceCurrentAlarmState := GVL_IO.aInputState[2].1;
				bDeviceCurrentWarningState := GVL_IO.aInputState[2].1;
			8: //DOR Fault
				bAlarmEnable := GVL_IO.aInterlockEnable[4].15;
				bWarningEnable := GVL_IO.aInterlockEnable[5].15;
				IF (GVL_IO.nDorOperationError = 1) THEN
					bDeviceCurrentAlarmState := TRUE;
				ELSE
					bDeviceCurrentAlarmState := FALSE;
				END_IF
				IF (GVL_IO.nDorOperationError = 2) OR (GVL_IO.nDorOperationError = 3) THEN
					bDeviceCurrentWarningState := TRUE;
				ELSE
					bDeviceCurrentWarningState := FALSE;
				END_IF
		END_CASE

		fbFaultCheck[i](
			bAlarmEnable := bAlarmEnable,
			bWarningEnable := bWarningEnable,
			bCurrentAlarmState := bDeviceCurrentAlarmState,
			bCurrentWarningState := bDeviceCurrentWarningState,
			tAlarmDelay := tAlarmDelay_D,
			bAlarm => bFaultAlarm,
			bWarning => bFaultWarning
			);
			
		IF bFaultAlarm THEN
			GVL_IO.aInterlock[1].0 := TRUE; //Alarm Trig
			GVL_IO.nCaseSignalTower := 1; // Signal Tower RED - Alarm
			//팝업 표시
			wAlarm := ROR(GVL_IO.aInterlock[2], (i+7));
			wAlarm.0 := TRUE;
			GVL_IO.aInterlock[2] := ROL(wAlarm, (i+7));
		END_IF
		IF bFaultWarning THEN
			GVL_IO.aInterlock[1].1 := TRUE; //Warning Trig
			GVL_IO.nCaseSignalTower := 2; // Signal Tower YELLOW - Warning
			//팝업 표시
			wAlarm := ROR(GVL_IO.aInterlock[4], (i+7));
			wAlarm.0 := TRUE;
			GVL_IO.aInterlock[4] := ROL(wAlarm, (i+7));
		END_IF
	END_FOR
	
	IF GVL_IO.aInterlockEnable[1].0 THEN //알람 리셋 버턴을 눌렀을 때
		GVL_IO.aInterlock[1].0 := FALSE; //Alarm Trig Reset
		GVL_IO.aInterlockEnable[1].0 := FALSE; //버턴 초기화
		GVL_IO.nCaseSignalTower := 4; // Signal Tower Blue - Idle
	END_IF
	IF GVL_IO.aInterlockEnable[1].1 THEN //주의 리셋 버턴을 눌렀을 때
		GVL_IO.aInterlock[1].1 := FALSE; //Warmomg Trig Reset
		GVL_IO.aInterlockEnable[1].1 := FALSE; //버턴 초기화
		GVL_IO.nCaseSignalTower := 4; // Signal Tower Blue - Idle
	END_IF	
END_IF

// bRecipeStartAvailable := //레시피 가능한 상태이면 TRUE
// 	NOT(AlarmTrig) AND
// 	NOT(WarningTrig) AND
// 	NOT(bMaintKey) AND
// 	GVL_IO.aInputState[2].4 AND //Cover Lower Limt
// 	GVL_IO.aInputState[4].6 AND //DOR State
// 	NOT(RCP.state_RcpOperation = 10) AND //Not Recipe Run State
// 	NOT(bGasStateProcess) AND //Safety Process Gas : TRUE
// 	NOT(bGasStateSource) AND //Safety Source Gas : TRUE
// 	NOT(bGasStateVent) AND
// 	P11_E3508.bManAuto_E3508 AND //Temperature Controller Auto : True
// 	P12_IQ_PLUS.ingPressureControl //Throttle Valve Pressure Control Mode : True 
// 	;
bRecipeStartAvailable := TRUE; // 테스트용 변수

bDorOnEnable :=
	NOT(AlarmTrig) AND
	GVL_IO.isCoverClosed AND
	GVL_IO.bDorState AND
	GVL_IO.isPumpRunning
	;
bHeaterOnEnable := bDorOnEnable;

// DOR Off Conditions
IF  GVL_IO.aController_PV[27] < GVL_IO.aInterlockSet[13] THEN
	bOpenEnableTemp := TRUE;
ELSE
	bOpenEnableTemp := FALSE;
END_IF
IF  GVL_IO.aController_PV[28] < GVL_IO.aInterlockSet[14] THEN
	bOpenEnablePress := TRUE;
ELSE
	bOpenEnablePress := FALSE;
END_IF
bDorOffEnable :=
	NOT(AlarmTrig) AND
	NOT(GVL_IO.bDORState) AND
	RCP.userState <> 10 AND //Not Recipe Run State
	bGasStateProcess AND //Safety Process Gas : TRUE
	bGasStateSource AND //Safety Source Gas : TRUE
	bGasStateVent AND //Vent Valve는 펌프 뒤쪽 Open
	GVL_IO.aInterlockEnable[6].4 AND //Can Open Temperature Check
	bOpenEnableTemp AND
	GVL_IO.aInterlockEnable[6].5 AND //Can Open Pressure Check
	bOpenEnablePress ;
GVL_IO.nUIInterockCheckOpenReactor.0 := NOT(AlarmTrig);
GVL_IO.nUIInterockCheckOpenReactor.1 := bOpenEnableTemp;
GVL_IO.nUIInterockCheckOpenReactor.2 := bOpenEnablePress;
GVL_IO.nUIInterockCheckOpenReactor.3 := NOT(GVL_IO.bDORState);
GVL_IO.nUIInterockCheckOpenReactor.4 := RCP.userState <> 10;
GVL_IO.nUIInterockCheckOpenReactor.5 := bGasStateProcess;
GVL_IO.nUIInterockCheckOpenReactor.6 := bGasStateSource;
GVL_IO.nUIInterockCheckOpenReactor.7 := bGasStateVent;
GVL_IO.nUIInterockCheckOpenReactor.8 := GVL_IO.aInterlockEnable[6].4;
GVL_IO.nUIInterockCheckOpenReactor.9 := GVL_IO.aInterlockEnable[6].5;
bReactorOpenEnable := bDorOffEnable;

(* Out to Device*)
GVL_IO.aDigitalOutputIO[3].7 := bPowerResetLED;
GVL_IO.aDigitalOutputIO[2].4 := bUPSMode;
GVL_IO.bDorOnEnable := bDorOnEnable;

END_PROGRAM

// ---- POUs/FB_DeviationCheck.TcPOU
//*********************************************************************
// Function Block: FB_DeviationCheck
// Description: 각 디바이스의 편차 초과 알람을 처리합니다.
// bEnable이 TRUE일 때만 알람 로직이 활성화됩니다.
//*********************************************************************
FUNCTION_BLOCK FB_DeviationCheck
VAR_INPUT
	bAlarmEnable	: BOOL; // 디바이스 활성화/비활성화 (TRUE = 활성화)
	bWarningEnable	: BOOL;
	fCurrentValue 	: REAL; //현재값
	fControlValue 	: REAL; //제어값
	fMaxValue		: REAL; //최대값
	fAlarmTreshold	: REAL; // 알람 편차 허용 임계값
	fWarningTreshold : REAL; // 경고 편차 허용 임계값
	tAlarmDelay		: TIME; //알람 지연 시간
END_VAR
VAR_OUTPUT
	bDeviationAlarm		: BOOL; //편차 알람 발생
	bDeviationWarning 	: BOOL; //편차 경고 발생
	fDeviationAlarm		: REAL; // 현재 편차(참고용)
	fDeviationWarning	: REAL; 
END_VAR
VAR
	// 내부 변수 (인스턴스별로 독립적)
	fbDeviationAlarmTimer 		: TON;
	fbDeviationWarningTimer 	: TON; 
	bDeviationAlarmCondition 	: BOOL;
	bDeviationWarningCondition 	: BOOL; 
END_VAR

// bAlarmEnable이 TRUE일 때만 알람 로직 실행
IF bAlarmEnable AND (fMaxValue <> 0) THEN
	fDeviationAlarm :=ABS(fCurrentValue - fControlValue)/fMaxValue * 100; //편차 계산(%)
	//편차 알람 로직(지연 시간 적용)
	IF fDeviationAlarm > fAlarmTreshold THEN
		bDeviationAlarmCondition := TRUE;
	ELSE
		bDeviationAlarmCondition := FALSE;
	END_IF
	fbDeviationAlarmTimer(IN:=bDeviationAlarmCondition, PT:=tAlarmDelay);
	bDeviationAlarm := fbDeviationAlarmTimer.Q;
ELSE
	// bEnable이 FALSE일 경우, 모든 알람 및 타이머를 비활성화/리셋
    // Q 출력을 FALSE로 강제하고, IN 입력을 FALSE로 설정하여 타이머를 리셋합니다.
	bDeviationAlarm := FALSE;
	fbDeviationAlarmTimer(IN := FALSE, PT := tAlarmDelay); // 타이머 리셋
	bDeviationAlarmCondition := FALSE; // 조건 플래그도 리셋
	fDeviationAlarm := 0.0; // 편차 값도 0으로 초기화 (선택 사항)
END_IF

// bWarningEnable이 TRUE일 때만 알람 로직 실행
IF bWarningEnable AND (fMaxValue <> 0) THEN
	//편차 계산(%)
	fDeviationWarning :=ABS(fCurrentValue - fControlValue)/fMaxValue * 100;
	//편차 알람 로직(지연 시간 적용)
	IF (fDeviationWarning > fWarningTreshold) AND (fDeviationWarning <= fAlarmTreshold) THEN
		bDeviationWarningCondition := TRUE;
	ELSE
		bDeviationWarningCondition := FALSE;
	END_IF
	fbDeviationWarningTimer(IN:=bDeviationWarningCondition, PT:=tAlarmDelay);
	bDeviationWarning := fbDeviationWarningTimer.Q;
ELSE
	// bEnable이 FALSE일 경우, 모든 알람 및 타이머를 비활성화/리셋
    // Q 출력을 FALSE로 강제하고, IN 입력을 FALSE로 설정하여 타이머를 리셋합니다.
	bDeviationWarning := FALSE;
	fbDeviationWarningTimer(IN := FALSE, PT := tAlarmDelay); // 타이머 리셋
	bDeviationWarningCondition := FALSE; // 조건 플래그도 리셋
	fDeviationWarning := 0.0; // 편차 값도 0으로 초기화 (선택 사항)
END_IF

END_FUNCTION_BLOCK

// ---- POUs/FB_SensorLimitCheck.TcPOU
//*********************************************************************
// Function Block: FB_SensorLimit
// Description: 각 디바이스의 범위 초과 알람을 처리합니다.
// bEnable이 TRUE일 때만 알람 로직이 활성화됩니다.
//*********************************************************************
FUNCTION_BLOCK FB_SensorLimitCheck
VAR_INPUT
	bAlarmEnable	: BOOL; //디바이스 활성화/비활성화 (TRUE = 활성화)
	bWarningEnable	: BOOL;
	fCurrentValue 	: REAL; //현재값
	fAlarmTreshold	: REAL; //알람 허용 임계값
	fWarningTreshold : REAL; //경고 허용 임계값
	tAlarmDelay		: TIME; //지연 시간
END_VAR
VAR_OUTPUT
	bLimitAlarm		: BOOL; //허용 값 초과 경고 발생
	bLimitWarning	: BOOL; //허용 값 초과 주의 발생
END_VAR
VAR
	// 내부 변수 (인스턴스별로 독립적)
	fbLimitAlarmTimer 		: TON;
	fbLimitWarningTimer 	: TON;
 	bLimitAlarmCondition 	: BOOL;
	bLimitWarningCondition 	: BOOL; 
END_VAR

// bAlarmEnable이 TRUE일 때만 알람 로직 실행
IF bAlarmEnable THEN
	//허용값 알람 로직(지연 시간 적용)
	IF fCurrentValue < fAlarmTreshold THEN
		bLimitAlarmCondition := TRUE;
	ELSE
		bLimitAlarmCondition := FALSE;
	END_IF
	fbLimitAlarmTimer(IN:=bLimitAlarmCondition, PT:=tAlarmDelay);
	bLimitAlarm := fbLimitAlarmTimer.Q;
ELSE
	// bEnable이 FALSE일 경우, 모든 알람 및 타이머를 비활성화/리셋
    // Q 출력을 FALSE로 강제하고, IN 입력을 FALSE로 설정하여 타이머를 리셋합니다.
	bLimitAlarm := FALSE;
	fbLimitAlarmTimer(IN := FALSE, PT := tAlarmDelay); // 타이머 리셋
	bLimitAlarmCondition := FALSE; // 조건 플래그도 리셋
END_IF

// bWarningEnable이 TRUE일 때만 알람 로직 실행
IF bWarningEnable THEN
	//허용값 주의 로직(지연 시간 적용)
	IF (fCurrentValue < fWarningTreshold) AND (fCurrentValue >= fAlarmTreshold ) THEN
		bLimitWarningCondition := TRUE;
	ELSE
		bLimitWarningCondition := FALSE;
	END_IF
	fbLimitWarningTimer(IN:=bLimitWarningCondition, PT:=tAlarmDelay);
	bLimitWarning := fbLimitWarningTimer.Q;
ELSE
	// bEnable이 FALSE일 경우, 모든 알람 및 타이머를 비활성화/리셋
    // Q 출력을 FALSE로 강제하고, IN 입력을 FALSE로 설정하여 타이머를 리셋합니다.
	bLimitWarning := FALSE;
	fbLimitWarningTimer(IN := FALSE, PT := tAlarmDelay); // 타이머 리셋
	bLimitWarningCondition := FALSE; // 조건 플래그도 리셋
END_IF

END_FUNCTION_BLOCK

// ---- POUs/FB_FaultCheck.TcPOU
//*********************************************************************
// Function Block: FB_FaultCheck
// Description: 각 디바이스의 Fault 발생시 알람을 처리합니다.
// bEnable이 TRUE일 때만 알람 로직이 활성화됩니다.
//*********************************************************************
FUNCTION_BLOCK FB_FaultCheck
VAR_INPUT
	bAlarmEnable		: BOOL; //디바이스 활성화/비활성화 (TRUE = 활성화)
	bWarningEnable		: BOOL;
	bCurrentAlarmState	: BOOL;
	bCurrentWarningState	: BOOL;
	tAlarmDelay			: TIME; //지연 시간
END_VAR
VAR_OUTPUT
	bAlarm		: BOOL; //허용 값 초과 경고 발생
	bWarning	: BOOL; //허용 값 초과 주의 발생
END_VAR
VAR
	// 내부 변수 (인스턴스별로 독립적)
	fbAlarmTimer 		: TON;
	fbWarningTimer 		: TON;
	bAlarmCondition 	: BOOL;
	bWarningCondition 	: BOOL; 
END_VAR

// bAlarmEnable이 TRUE일 때만 알람 로직 실행
IF bAlarmEnable THEN
	//허용값 알람 로직(지연 시간 적용)
	IF bCurrentAlarmState THEN
		bAlarmCondition := TRUE;
	ELSE
		bAlarmCondition := FALSE;
	END_IF
	fbAlarmTimer(IN:=bAlarmCondition, PT:=tAlarmDelay);
	bAlarm := fbAlarmTimer.Q;
ELSE
	// bEnable이 FALSE일 경우, 모든 알람 및 타이머를 비활성화/리셋
    // Q 출력을 FALSE로 강제하고, IN 입력을 FALSE로 설정하여 타이머를 리셋합니다.
	bAlarm := FALSE;
	fbAlarmTimer(IN:=FALSE, PT:= tAlarmDelay); // 타이머 리셋
	bAlarmCondition := FALSE; // 조건 플래그도 리셋
END_IF

// bWarningEnable이 TRUE일 때만 알람 로직 실행
IF bWarningEnable THEN
	//허용값 알람 로직(지연 시간 적용)
	IF bCurrentWarningState THEN
		bWarningCondition := TRUE;
	ELSE
		bWarningCondition := FALSE;
	END_IF
	fbWarningTimer(IN:=bWarningCondition, PT:=tAlarmDelay);
	bWarning := fbWarningTimer.Q;
ELSE
	// bEnable이 FALSE일 경우, 모든 알람 및 타이머를 비활성화/리셋
    // Q 출력을 FALSE로 강제하고, IN 입력을 FALSE로 설정하여 타이머를 리셋합니다.
	bWarning := FALSE;
	fbWarningTimer(IN:=FALSE, PT:= tAlarmDelay); // 타이머 리셋
	bWarningCondition := FALSE; // 조건 플래그도 리셋
END_IF

END_FUNCTION_BLOCK

// ---- FUNTION/Real_To_String_LineHeater.TcPOU
FUNCTION Real_To_String_LineHeater : STRING
VAR_INPUT
	rTemperatureSV 		: REAL;
	nHeaterNumber		: INT;
END_VAR
VAR
	wTemperature		: WORD;
	hStrTemp			: STRING;
	sHeaterNumber		: STRING;
	sString				: STRING;
	sSendString			: STRING;
END_VAR

//LH: Line Heater x 8EA -> 8Channel TIC 1EA
//Model: HANYOUNG NUX, MC9-8RD0SS32

// Multiple decimal place point
// STRING : '$0201DWR,03,0301(ZONE_NO),0001(ZONE_1),0302(CH_NO),0001(CH_1,sHeaterNumber),0401(SV), hStrTemp, $0D$0A'
sString := '$0201DWR,03,0301,0001,0302,,0401,,$0D$0A';

//Convert to Channel from Heater Number
sHeaterNumber := DINT_TO_DECSTR(nHeaterNumber, 4);
sString := INSERT(sString,sHeaterNumber,25);
	
//Convert to String Type
wTemperature := REAL_TO_WORD(rTemperatureSV);
hStrTemp := WORD_TO_HEXSTR(wTemperature, 4, FALSE);
Real_To_String_LineHeater := INSERT(sString,hStrTemp,35);

END_FUNCTION

// ---- POUs/P14_ThermalBath.TcPOU
PROGRAM P14_ThermalBath
VAR
	rTemperatureSV 		: ARRAY[1..6]OF REAL;

	(* Input from Device *)
	bTempDeviationAlarm	: ARRAY[1..6] OF BOOL;
	bCutOffAlarm		: ARRAY[1..6] OF BOOL;
	
	rTemperature_PV 		: ARRAY[1..6]OF REAL;
	isBath_Err 			: ARRAY[1..6]OF BOOL;
	isBath_TC_Broken 	: ARRAY[1..6]OF BOOL ; 

	//for send variable
	TimeOnDelay	: TON; //Time delay after Power ON of Thermal Bath
	TimeCycle			: TON;
	TimeWaitSend		: TON;
	TimeWaitReceive		: TON;
	bSendingEnable 		: BOOL:=TRUE; // Check the Sending Stage
	bSetValueMode 		: BOOL;
	rTemperatureTV 		: ARRAY[1..6]OF REAL;
	fbSend				: SendString;
	sSendString 		: STRING;
	bSendBusy			: BOOL;
	bSendingOK 			: BOOL;
	eSendErrorID		: ComError_t;

	// for received variable
	fbReceive			: ReceiveString;
	sReceivedString		: STRING;
	bStringReceived		: BOOL;
	bReceiveBusy		: BOOL;
	bReceiveError		: BOOL;
	eReceiveErrorID		: ComError_t;
	bReceiveTimeout		: BOOL;
	bReceivedOK 		: BOOL;
	
	nBathNumber 		: INT := 1;
	sBathNumber 		: STRING := '1';
	sReceivedBathNumber : STRING;
	nReceivedBathNumber : INT;
	sReceivedAffirmation : STRING;
	sReceivedData 		: STRING;
	
	(* Input *)
	bThermalBathCB		: BOOL;
	index				: INT;
END_VAR

// Call the send block every second to repeat the transmission.
// Also call the block as long as it is busy to finish a transmission.
//TB: Thermal Bath x 6EA
//Maker: SMC
//Model: HEBC002-WA10
//Temp Range: -15 ~60℃
//RS485: 9600, DataBit(8), Parity(None), StopBit(1)
//BCC Check X

(* Read from Power Distribution Pannel *)
bThermalBathCB := GVL_IO.aDigitalInputIO[5].0;

(* Read from SMC Bath Device Value *)
TimeOnDelay(IN:= P90_Interlock.bThermalBathMC, PT :=T#1S); //Time Delay after a Thermal Bath MC ON
bTempDeviationAlarm[1]	:= GVL_IO.aDigitalInputIO[8].0;
bTempDeviationAlarm[2]	:= GVL_IO.aDigitalInputIO[8].2;
bTempDeviationAlarm[3]	:= GVL_IO.aDigitalInputIO[8].4;
bTempDeviationAlarm[4]	:= GVL_IO.aDigitalInputIO[8].6;
bTempDeviationAlarm[5]	:= GVL_IO.aDigitalInputIO[9].0;
bTempDeviationAlarm[6]	:= GVL_IO.aDigitalInputIO[9].2;
bCutOffAlarm[1] := NOT(GVL_IO.aDigitalInputIO[8].1); //Normally Contact
bCutOffAlarm[2] := NOT(GVL_IO.aDigitalInputIO[8].3);
bCutOffAlarm[3] := NOT(GVL_IO.aDigitalInputIO[8].5);
bCutOffAlarm[4] := NOT(GVL_IO.aDigitalInputIO[8].7);
bCutOffAlarm[5] := NOT(GVL_IO.aDigitalInputIO[9].1);
bCutOffAlarm[6] := NOT(GVL_IO.aDigitalInputIO[9].3);

// make a sending string
TimeCycle(IN := TimeOnDelay.Q, PT := T#1S); //Cycle for Serial Communication
IF TimeCycle.Q = TRUE THEN
	TimeCycle(IN := FALSE);

	// Make a sending string Set value or Request value 
	IF bSendingEnable = TRUE THEN
		//Set sate
		bSendingEnable := FALSE;
		bReceivedOK := FALSE;
		bSetValueMode := FALSE;
		
		//Target value(Bath) Set value
		IF (rTemperatureTV[nBathNumber] <> rTemperatureSV[nBathNumber])  OR isBath_Err[nBathNumber] THEN
			rTemperatureTV[nBathNumber] := rTemperatureSV[nBathNumber];
			sSendString := Real_To_String_ThermalBath(rTemperatureTV[nBathNumber],nBathNumber); //Send a SetValue=10.0 '$0201WSV100100$03'
			bSetValueMode := TRUE;
		ELSE
			sBathNumber := INT_TO_STRING(nBathNumber);
			sSendString := INSERT('$020RPV1$03',sBathNumber,2); //Request a PV
			bSetValueMode := FALSE;
		END_IF
		
		// Send string	
		fbSend(	SendString:= sSendString,
			TXbuffer:= TxBufferTB,
			Busy=> bSendBusy,
			Error=> );
		IF fbSend.Error <> COMERROR_NOERROR THEN
			eSendErrorID := fbSend.Error;
			bSendingOK := FALSE;
		ELSE
			eSendErrorID := COMERROR_NOERROR;
			bSendingOK := TRUE;
		END_IF
		
	END_IF

	//	Receive string data:
	//	The block receives any data strings beginning with a STX ($02) and ending with an ETX ($03) character.
	TimeWaitReceive(IN := bSendingOK, PT := T#250MS); //Wait receiving data
	IF TimeWaitReceive.Q THEN
		TimeWaitReceive(IN:= FALSE);
		fbReceive(
			Prefix:= '$02',
			Suffix:= '$03',
			Timeout:= T#1S,
			ReceivedString:= sReceivedString,
			RXbuffer:= RxBufferTB,
			StringReceived=> bStringReceived,
			Busy=> bReceiveBusy,
			Error=> ,
			RxTimeout=> bReceiveTimeout );
			
		IF bReceiveTimeout THEN
			isBath_Err[nReceivedBathNumber] := TRUE;
			bReceiveTimeout := FALSE;
		END_IF
		
		IF fbReceive.Error <> COMERROR_NOERROR THEN
			eReceiveErrorID := fbReceive.Error;
		END_IF
		
		IF bStringReceived THEN
			bStringReceived :=FALSE;
			bReceivedOK := TRUE;
			bSendingEnable := TRUE;
			sReceivedBathNumber := MID(STR:=sReceivedString, len:=1, pos:=3); //ReceivedString : '$0201$06PV100250$03'
			nReceivedBathNumber := STRING_TO_INT(sReceivedBathNumber);
			sReceivedAffirmation := MID(STR:=sReceivedString, len:=1, pos:=4); //Affirmation
			
			IF bSetValueMode THEN //Write SV Mode
				IF sReceivedAffirmation = '$06' THEN //'$06' ReceivedString : '$0201$06$03'
					isBath_Err[nReceivedBathNumber] := FALSE;
				ELSE
					//isBath_Err[nReceivedBathNumber] := TRUE;
				END_IF
				bSetValueMode := FALSE;
			ELSE //Read PV Mode
				sReceivedData := MID(STR:=sReceivedString, len:=5, pos:=8); //ReceivedString : '$0201$06PV100250$03'
				IF sReceivedData = '' THEN
					//isBath_Err[nReceivedBathNumber] := TRUE;
				ELSIF sReceivedData = 'HHHHH' THEN
					rTemperature_PV[nReceivedBathNumber] := -99.0;
					isBath_TC_Broken[nReceivedBathNumber] := TRUE;
					isBath_Err[nReceivedBathNumber] := FALSE;
				ELSE
					rTemperature_PV[nReceivedBathNumber] := (STRING_TO_REAL(sReceivedData))/10;
					isBath_TC_Broken[nReceivedBathNumber] := FALSE;
					isBath_Err[nReceivedBathNumber] := FALSE;
				END_IF
			END_IF
			index := nReceivedBathNumber + 11;
			GVL_IO.aMonitoring_PV[index] := rTemperature_PV[nReceivedBathNumber];
			
		END_IF
	END_IF
	
	//Change the Next Bath
	nBathNumber := nBathNumber + 1;
	IF nBathNumber > 6 THEN
		nBathNumber := 1;
	END_IF
	bSendingEnable := TRUE;
END_IF

END_PROGRAM

// ---- FUNTION/Real_To_String_ThermalBath.TcPOU
FUNCTION Real_To_String_ThermalBath : STRING
VAR_INPUT
	rTemperatureSV 	: REAL;
	nBathNumber		: INT;
END_VAR
VAR
	sBathNumber 	: STRING;
	rTemp 			: REAL;
	nTemp 			: DINT;
	sTemp 			: STRING;
	sBaseString		: STRING;
END_VAR

// Thermal Bath SMC HEBC002-WA10
rTemp := rTemperatureSV*10 ;
nTemp := REAL_TO_DINT(rTemp);
sBaseString := '$020WSV1$03';

sBathNumber := INT_TO_STRING(nBathNumber);
sBaseString := INSERT(sBaseString,sBathNumber,2);

IF nTemp >= 0 THEN
	sTemp := DINT_TO_DECSTR(nTemp, 5); //00010
ELSE
	sTemp := DINT_TO_DECSTR(nTemp, 4); 
	sTemp := CONCAT('-',sTemp); //-0010
END_IF

sBaseString := INSERT(sBaseString,sTemp,7);

Real_To_String_ThermalBath := sBaseString;

END_FUNCTION

// ---- POUs/P15_RotationOperation.TcPOU
PROGRAM P15_RotationOperation
VAR
	rControlValue			: REAL; //rpm
	bAlarmReset				: BOOL; //Motor Driver Alarm

	bRotationCP				: BOOL;
	nConvertedRotation_PV	: INT; //PV 0~100 rpm

	rConvertedCV			:REAL;
	(* Motor Driver *)
	bBrake_Run				: BOOL;
	(* Rotation Operation Parameter*)
	wRotaion_PV				: WORD;
	isRotationFault			: BOOL; //Motor Driver
END_VAR

VAR CONSTANT
	KL4404MaxValueP		: REAL := 13106; //0~4V, 0~2500RPM, BLHM230K-GFS
	//Motor Max Rotation RPM 2,500rpm, Gear Ratio 15, Belt Ratio 1.5
	ConversionFactor 	: REAL :=117.9585; //KL4404MaxValueP*15*1.5/2500
END_VAR

// Oriental Motor Driver : BLHM230K-GFS, 0~4V

(* Read from Power Distribution Pannel *)
bRotationCP := GVL_IO.aDigitalInputIO[5].3;

//from Device Value
isRotationFault := NOT(GVL_IO.aDigitalInputIO[2].5);
wRotaion_PV := UINT_TO_WORD(GVL_IO.aAnalogInputIO2[1]);
nConvertedRotation_PV := REAL_TO_INT(wRotaion_PV/(5*ConversionFactor));

// Interface with other PRGs
GVL_IO.nRotation_Converted_PV := nConvertedRotation_PV;
rControlValue := LREAL_TO_REAL(GVL_IO.aController[29].rControlValue);

//Write to Motor Driver
rConvertedCV := rControlValue * ConversionFactor; // Convert from RPM to control value

IF (GVL_IO.aController[29].input.targetValue > 0) OR (wRotaion_PV > 0) THEN // Motor Driver RUN
	bBrake_Run := TRUE;
ELSIF (GVL_IO.aController[29].input.targetValue = 0) AND (wRotaion_PV = 0) THEN
	bBrake_Run := FALSE;
END_IF

GVL_IO.aDigitalOutputIO[3].4 	:= bBrake_Run;
GVL_IO.aDigitalOutputIO[3].5 	:= bBrake_Run;
GVL_IO.aAnalogOutputIO[28] 		:= REAL_TO_INT(rConvertedCV);
GVL_IO.aInputState[1].11		:= isRotationFault;

END_PROGRAM

// ---- POUs/P16_CoverOperation.TcPOU
PROGRAM P16_CoverOperation
VAR
// 	isCoverClosed 	: BOOL;

	bCoverCP	: BOOL;
	bLowerLimit	: BOOL;
	bUpperLimit	: BOOL;
	TimerUpLED 		: TON;
	TimerUpLED_X 	: TON;
	TimerDownLED 	: TON;
	TimerDownLED_X 	: TON;
	TimerDownDelayOff 	: TON;
	(* Input *)
	bUpSwitch	: BOOL;
	bDownSwitch 	: BOOL;
	(* Output *)
	bUpLED 		: BOOL;
	bDownLED 	: BOOL;
	bOnUpRelay 	: BOOL;
	bOnDownRelay : BOOL;		
END_VAR

(* Read from Device Value *)
// Cover Operation Switch
bUpSwitch 		:= GVL_IO.aDigitalInputIO[1].6;
bDownSwitch 	:= GVL_IO.aDigitalInputIO[1].7;
bUpperLimit 	:= GVL_IO.aDigitalInputIO[3].4;
bLowerLimit 	:= GVL_IO.aDigitalInputIO[3].5;
bCoverCP 		:=  GVL_IO.aDigitalInputIO[5].4;

TimerDownDelayOff(IN:=bLowerLimit, PT:=T#500MS);

// Cover Operation Condition
IF P90_Interlock.bReactorOpenEnable THEN
	bOnUpRelay := (bDownSwitch = FALSE AND bUpSwitch = TRUE AND bUpperLimit = FALSE);
	bOnDownRelay := (bDownSwitch = TRUE AND bUpSwitch = FALSE AND (bLowerLimit = FALSE OR TimerDownDelayOff.Q = FALSE ));
END_IF

//LED Blinking
TimerUpLED(IN:=(bOnUpRelay AND TimerUpLED_X.Q = FALSE), PT:=T#500MS);
TimerUpLED_X(IN:=TimerUpLED.Q, PT:=T#300MS);
bUpLED := (TimerUpLED.Q AND bOnUpRelay) OR bUpperLimit;

TimerDownLED(IN:=(bOnDownRelay AND TimerDownLED_X.Q = FALSE), PT:=T#500MS);
TimerDownLED_X(IN:=TimerDownLED.Q, PT:=T#300MS);
bDownLED := (TimerDownLED.Q AND bOnDownRelay) OR bLowerLimit;

//Status Output
GVL_IO.isCoverClosed := bLowerLimit;

(* Write to Device Value *)
// Cover Operation Switch Lamp
GVL_IO.aDigitalOutputIO[4].2 := bUpLED;
GVL_IO.aDigitalOutputIO[4].3 := bDownLED;
GVL_IO.aDigitalOutputIO[1].6 := bOnUpRelay;
GVL_IO.aDigitalOutputIO[1].7 := bOnDownRelay;

END_PROGRAM

// ---- POUs/P17_DOROperation.TcPOU
PROGRAM P17_DOROperation
VAR
	bDOROn				: BOOL; //UI Input Button
	bDOROff				: BOOL; //UI Input Button
	fTresholdPressure	: REAL;
	fTresholdCount		: REAL;
	bPressureEnable 	: BOOL;
	bCountEnable		: BOOL;

	isDOROnState		: BOOL := FALSE; //DOR ON State
	bError				: INT; //0: No Err, 1: Vacuum Fail, 2: Vacuum Release, 3: Try out
	nWaitCounter		: INT;

	(* Input *)
	bVacSwitch			: BOOL; //Push Switch
	bAtmSwitch			: BOOL; //Push Switch
	(* Pressure Transducer *)
	nPressurePV			: INT;
	rPressurePV_kPa		: REAL;
	(* Output *)
	bVacLED				: BOOL;
	bAtmLED				: BOOL;
	bV_DORVac			: BOOL; //V34 Valve
	bV_DORFill			: BOOL; //V35 Valve
	
	(* DOR Condition Operation Parameter *)
	rTrigSwitch			: R_TRIG;
	TimerOnLED			: TON;
	TimerVacSwitch		: TON;
	TimerAtmSwitch		: TON;
	TimerWaitCheck		: TON;
	TimerVacRealease	: TON;
	nCase				: INT := 0;
	nTresholdCount		: INT;
	nTryCount			: INT;
	bVacuumRealse		: BOOL;
	//Temperatur Variable
	bTest				: BOOL;
	nTest				: INT;
END_VAR

VAR CONSTANT
	KL3464MaxValueP		: REAL := 16383; //1 ~ 5VDC, 0 ~ 100kPa(1bar), PG35
	SlopeFactor			: REAL := 0.007617887; //100kPa/(16383-3256)
END_VAR

// Double O-Ring Vacuum Condition

(* Read from Device Value *)
// DOR Operation Switch
bVacSwitch 			:= GVL_IO.aDigitalInputIO[1].4; //Switch Input
bAtmSwitch 			:= GVL_IO.aDigitalInputIO[1].5; //Switch Input
nPressurePV 		:= GVL_IO.aAnalogInputIO[29];
rPressurePV_kPa 	:= (nPressurePV-3256)*SlopeFactor;

fTresholdPressure 	:= GVL_IO.aInterlockSet[15];
fTresholdCount 		:= GVL_IO.aInterlockSet[16];
bPressureEnable 	:= GVL_IO.aInterlockEnable[1].5;
bCountEnable 		:= GVL_IO.aInterlockEnable[1].6;
nTresholdCount 		:= REAL_TO_INT(fTresholdCount); //Try One more Vacuum 

(* If Vacuum 'ON' Switch Press, Change DOR Vacuum State *)
//DOR Operation Signal generation
TimerVacSwitch(IN:=bVacSwitch OR bDOROn, PT:=T#100MS);
rTrigSwitch(CLK:=TimerVacSwitch.Q);

IF rTrigSwitch.Q AND GVL_IO.bDorOnEnable THEN
	nCase 		:= 1;
	nTryCount 	:= 1; //Try One more Vacuum 
END_IF

CASE nCase OF
	1: //Initialize
		isDOROnState := FALSE;
		bV_DORVac 	:= TRUE; //V34 Open
		bV_DORFill	:= FALSE; //V35 Close
		bAtmLED		:= FALSE;
		TimerWaitCheck(IN:=FALSE);	
		nCase := 10;
	10: //Wait and Vacuum Check
		(* Blink Switch LED *)
		TimerOnLED(IN:=TRUE, PT:=T#500MS);
		IF TimerOnLED.Q THEN
			TimerOnLED(IN:=FALSE);
			bVacLED := NOT(bVacLED);
		END_IF

		TimerWaitCheck(IN:=TRUE, PT:=T#5S);
		IF TimerWaitCheck.Q THEN
			IF rPressurePV_kPa > fTresholdPressure THEN
				bV_DORVac 		:= FALSE; //V34 Close
				isDOROnState 	:= TRUE;
				bVacLED 		:= TRUE; //Switch LED
				bError			:= 0;
				nCase 			:= 0;
			ELSIF nTryCount < nTresholdCount THEN
				TimerWaitCheck(IN:=FALSE);
				nTryCount 		:= nTryCount + 1;				
				nCase 			:= 1;
			ELSE
				bV_DORVac 		:= FALSE; //V34 Close
				isDOROnState 	:= FALSE;
				bVacLED			:= FALSE; //Switch LED
				bError			:= 1; // Vacuum Fail
				nCase			:= 0;
			END_IF
		END_IF
END_CASE

(* If Vacuum 'OFF' Switch Press, Change DOR Vent(Fill, Atm) State *)
//DOR Operation Signal generation
TimerAtmSwitch(IN:=bAtmSwitch OR bDOROff, PT:=T#100MS);
rTrigSwitch(CLK:=TimerAtmSwitch.Q);

IF rTrigSwitch.Q AND P90_Interlock.bDorOffEnable THEN
	nCase := 2;
END_IF

CASE nCase OF
	2:
		(* Blink Switch LED *)
		TimerOnLED(IN:=TRUE, PT:=T#500MS);
		IF TimerOnLED.Q THEN
			TimerOnLED(IN:=FALSE);
			bAtmLED := NOT(bAtmLED);
		END_IF
		
		TimerWaitCheck(IN:=TRUE, PT:=T#10S);
		nWaitCounter := TIME_TO_INT(TimerWaitCheck.ET/1000);
		IF TimerWaitCheck.Q THEN
			TimerWaitCheck(IN:=FALSE);
			bVacLED			:= FALSE;
			bV_DORVac 		:= FALSE; //V34 Close
			bV_DORFill		:= TRUE; //V35 Open
			nCase			:= 20;
		END_IF
	20:
		TimerWaitCheck(IN:=TRUE, PT:=T#5S);
		IF TimerWaitCheck.Q THEN
			bVacLED			:= FALSE;
			bV_DORFill		:= FALSE;
			isDOROnState 	:= FALSE;
			bAtmLED			:= TRUE;
			nCase			:= 0;
		END_IF
END_CASE

(* If Vacuum 'ON' State, Check the Vacuum range *)
IF isDOROnState AND rPressurePV_kPa < (fTresholdPressure - 20) AND nTryCount < 3 THEN
	bError := 2; // Vacuum release
	TimerVacRealease(IN:=TRUE, PT:=T#2S);
	
	(* Blink Vac Switch LED *)
	TimerOnLED(IN:=TRUE, PT:=T#500MS);
	IF TimerOnLED.Q THEN
		TimerOnLED(IN:=FALSE);
		bVacLED := NOT(bVacLED);
	END_IF

	IF TimerVacRealease.Q  THEN
		TimerVacRealease(IN:=FALSE);
		nTryCount 		:= nTryCount + 1;
		bV_DORVac 		:= FALSE;//Vacuum Valve OFF
		bVacLED := TRUE;
	ELSE
		bV_DORVac 		:= TRUE;//Vacuum Valve ON
	END_IF
	
ELSIF bError = 2 THEN
	bV_DORVac := FALSE;
	bError := 0;
	
ELSIF nTryCount >= 3 THEN
	bV_DORVac := FALSE;
	bError := 3; //Vacuum Released
END_IF

//알람 리셋
IF GVL_IO.aInterlockEnable[1].0 OR GVL_IO.aInterlockEnable[1].1 THEN
	bError := 0;
END_IF

(* Write to Device Value *)
// Cover Operation Switch Lamp
GVL_IO.aOutputSolValve[2].18 := bV_DORVac; //V34
GVL_IO.aOutputSolValve[2].19 := bV_DORFill; //V35
GVL_IO.aDigitalOutputIO[4].0 := bVacLED;
GVL_IO.aDigitalOutputIO[4].1 := bAtmLED;

GVL_IO.nDorOperationError := bError;
GVL_IO.bDorState := isDOROnState;

END_PROGRAM

// ---- POUs/P21_Background_LineHeater.TcPOU
PROGRAM P21_Background_LineHeater
VAR
	(* background communication with the KL6031 terminal (22byte)
	Thermal Bath(HEBC002-WA10) x 6EA *)
	fbCtrl		: SerialLineControl;
	bCtrlError	: BOOL;
	eCtrlErrorID	: ComError_t;
	fbConfig		: KL6configuration;
	bConfigError	: BOOL;
	eConfigErrorID: ComError_t;
	bConfigExe	: BOOL := TRUE;
	(* 	I/O variables for a KL6031 terminal*)	
	stIn_KL6031_LH AT %I*	: KL6inData22B;	(* linked to the KL6001 in the TwinCAT System Manager *)
	stOut_KL6031_LH AT %Q*	: KL6outData22B;	(* linked to the KL6001 in the TwinCAT System Manager *)
END_VAR

(*
The SerialLineControl function block is supposed to be called in every PLC cycle.
It communicates with the serial line hardware device and transmits or receives data.
The SerialLineControl can be called in the standard task (e.g.for PcCOM port usage) 
or in a separate fast task (e.g.for terminal usage) as well.
A fast separate task will be necessary at high baud rates or with KL6001 terminals 
which have a small process image (3 or 5 data bytes only)
Line Heater x 8EA -> 8Channel TIC 1EA
Maker: HANYOUNG NUX
Model: MC9-8RD0SS32
Temp Range: -15 ~200℃
RS485: 9600, DataBit(8), Parity(None), StopBit(1)
BCC Check X
*)

fbCtrl(
	Mode:= SERIALLINEMODE_KL6_22B_STANDARD,
	pComIn:= ADR(stIn_KL6031_LH),
	pComOut:= ADR(stOut_KL6031_LH),
	SizeComIn:= SIZEOF(stIn_KL6031_LH),
	Error=> ,
	ErrorID=> ,
	TxBuffer:= TxBufferLH,
	RxBuffer:= RxBufferLH );
IF fbCtrl.Error THEN
	bCtrlError := TRUE;
	eCtrlErrorID := fbCtrl.ErrorID;
END_IF

END_PROGRAM

// ---- POUs/P30_ManualControl.TcPOU
Program P30_ManualControl
VAR
	analogDeviceRampControl : FB_AnalogDeviceRampControl;
END_VAR

analogDeviceRampControl();

END_PROGRAM

// ---- POUs/FB_AnalogDeviceRampControl.TcPOU
FUNCTION_BLOCK FB_AnalogDeviceRampControl
VAR
	i : UINT;
END_VAR

FOR i:=1 TO GVL_IO.NumFlowController DO
	GVL_IO.aAnalogOutputIO[i] := LREAL_TO_INT(GVL_IO.aController[i].rControlValue / GVL_IO.AnalogControllerOutputVoltage * GVL_IO.KL3464MaxValueH);
	GVL_IO.aController[i]();
END_FOR

IF ( GVL_IO.aController[27].rControlValue > GVL_IO.TempDigitOutputFallbackThres ) THEN
	GVL_IO.aDigitalOutputIO[2].0 := TRUE;
ELSE
	GVL_IO.aDigitalOutputIO[2].0 := FALSE;
END_IF

GVL_IO.aController[27]();
GVL_IO.aController[28]();
GVL_IO.aController[29]();

END_FUNCTION_BLOCK

// ---- POUs/P50_RecipeControl.TcPOU
PROGRAM P50_RecipeControl
VAR
	nRcpIndex		: INT;
	eRecipeRun		: E_RecipeRun ; //레시피 상태
	fbAnalogDeviceRampControl : FB_AnalogDeviceRampControl;
	fbRecipeAnalogInputControlSequencer: FB_RecipeAnalogControlInputSequencer;
	fbValveControl: FB_ValveControl;
	
	Pause_TON		: TON;
	Ramp_TON		: FB_TON_Pausable;
	Hold_TON		: FB_TON_Pausable;
	
	loopCount		: ARRAY[1..100] OF INT;
	i				: INT;
	TotalETLast			: TIME := T#0S;
END_VAR
VAR CONSTANT
	Pause_MAX		: TIME := T#1800S;
END_VAR

CASE RCP.cmd_RcpOperation OF
	0: //Init State
 		f_ResetTimersAndRCPTimes(fbPause_TON := Pause_TON, fbRamp_TON := Ramp_TON, fbHold_TON := Hold_TON);
		TotalETLast := T#0S;
		RCP.TotalET := T#0S;
		
		FOR i:=1 TO Rcp.iRcpTotalStep DO
			loopCount[i] := Rcp.aRecipe[i].iRecipe[9];
		END_FOR
		
		nRcpIndex := 0;
		Rcp.userState := 0;
		eRecipeRun := E_RecipeRun.Initial;
		GVL_IO.nCaseSignalTower := 5; // White - Idle

	10: //RUN
		IF nRcpIndex = 0 THEN
			nRcpIndex := 1;
		END_IF
		fbAnalogDeviceRampControl();
						
		// CASE 문을 이용한 상태 머신 구현
		CASE eRecipeRun OF
			E_RecipeRun.Initial:
				f_ResetTimersAndRCPTimes(fbPause_TON := Pause_TON, fbRamp_TON := Ramp_TON, fbHold_TON := Hold_TON);
				fbRecipeAnalogInputControlSequencer(rRecipe := RCP.aRecipe[nRcpIndex].rRecipe, rampTime:= TO_UINT(RCP.aRecipe[nRcpIndex].iRecipe[2]), tempRecipe := TO_REAL(RCP.aRecipe[nRcpIndex].iRecipe[4]),
					pressRecipe := TO_REAL(RCP.aRecipe[nRcpIndex].iRecipe[5]), rotRecipe := TO_REAL(RCP.aRecipe[nRcpIndex].iRecipe[6]));
				fbValveControl(valveSetting:= RCP.aRecipe[nRcpIndex].dRecipe);
				Rcp.userState := 10;// Recipe Running
				GVL_IO.nCaseSignalTower := 3;
				eRecipeRun := E_RecipeRun.Ramp;
				
			E_RecipeRun.Ramp: // Ramp 수행
				Ramp_TON(IN:=TRUE, PT:= RCP.aRecipe[nRcpIndex].iRecipe[2] * T#1S, ET=>RCP.RecipeRunET.ET);
				RCP.TotalET := TotalETLast + RCP.RecipeRunET.ET;
				RCP.RecipeRunET.Mode := E_RecipeRunETMode.Ramp;
				IF Ramp_TON.Q THEN
					Ramp_TON(IN:=FALSE);
					eRecipeRun := E_RecipeRun.CheckHoldTemp;
					TotalETLast := RCP.TotalET;
				END_IF				
				
			E_RecipeRun.CheckHoldTemp: //Hold Temp 확인
				IF RCP.aRecipe[nRcpIndex].iRecipe[7] = 0 THEN
					Hold_TON(IN:=TRUE, PT:= RCP.aRecipe[nRcpIndex].iRecipe[3] * T#1S, ET=>RCP.RecipeRunET.ET);
					RCP.TotalET := TotalETLast + RCP.RecipeRunET.ET;
					RCP.RecipeRunET.Mode := E_RecipeRunETMode.Hold;
					IF Hold_TON.Q THEN
						Hold_TON(IN:=FALSE);
						TotalETLast := RCP.TotalET;
						eRecipeRun := E_RecipeRun.End; // 레시피 첫 Column 실행
					END_IF
				ELSIF GVL_IO.aController_PV[27] < RCP.aRecipe[nRcpIndex].iRecipe[7] THEN //서셉터 온도가 Wait 온도보다 낮을 때
					Hold_TON(IN:=FALSE);
					TotalETLast := RCP.TotalET;
					eRecipeRun := E_RecipeRun.End; // 레시피 첫 Column 실행
				ELSE // 서셉터 온도가 Wait 온도보다 높을 때
					;// 떨어질 때까지 기다림
				END_IF
				
			E_RecipeRun.End: // 다음 Step 이동 (루프 마지막 단계일 경우, 다음 Step 이동 또는 루프 처음단계로 점프)
				loopCount[nRcpIndex] := loopCount[nRcpIndex] - 1;
				nRcpIndex := nRcpIndex + 1 - (RCP.aRecipe[nRcpIndex].iRecipe[8]) * MIN(loopCount[nRcpIndex], 1);
				IF nRcpIndex > Rcp.iRcpTotalStep THEN
					RCP.cmd_RcpOperation := 50;
				END_IF
				eRecipeRun := E_RecipeRun.Initial;
		END_CASE
		
	20: //PAUSE
		CASE eRecipeRun OF
			E_RecipeRun.Ramp:
				Ramp_TON(PAUSE:=TRUE);		
			E_RecipeRun.CheckHoldTemp:
				Hold_TON(PAUSE:=TRUE);
		END_CASE
		
		Pause_TON(IN:=TRUE, PT:= Pause_MAX, ET=>RCP.Pause_ET); //최대 홀드 시간이 지나면 다음 스텝으로 넘거감
		IF Pause_TON.Q THEN
			Pause_TON(IN:=FALSE);
			eRecipeRun := E_RecipeRun.End; // 레시피 첫 Column 실행
		END_IF

		Rcp.userState := 20;
		GVL_IO.nCaseSignalTower := 5;
		
	30: //RESTART
		Pause_TON(IN:=FALSE);
		CASE eRecipeRun OF
			E_RecipeRun.Ramp:
				Ramp_TON(PAUSE:=FALSE);
			
			E_RecipeRun.CheckHoldTemp:
				Hold_TON(PAUSE:=FALSE);
		END_CASE

		RCP.Pause_ET := T#0S;
		Rcp.userState := 10;
		RCP.cmd_RcpOperation := 10;	
		GVL_IO.nCaseSignalTower := 3;
		
	40: //STOP
		f_ResetTimersAndRCPTimes(fbPause_TON := Pause_TON, fbRamp_TON := Ramp_TON, fbHold_TON := Hold_TON);
		TotalETLast := T#0S;
		RCP.TotalET := T#0S;
		Rcp.userState := 40;
		GVL_IO.nCaseSignalTower := 5;
		
	50: //END
		f_ResetTimersAndRCPTimes(fbPause_TON := Pause_TON, fbRamp_TON := Ramp_TON, fbHold_TON := Hold_TON);
		TotalETLast := T#0S;
		RCP.TotalET := T#0S;
		Rcp.userState := 50;
		fbAnalogDeviceRampControl();
		GVL_IO.nCaseSignalTower := 5;
		
	60: //SKIP
		IF E_RecipeRun.Ramp <= eRecipeRun  AND  eRecipeRun <= E_RecipeRun.CheckHoldTemp THEN
			eRecipeRun := E_RecipeRun.End;
		END_IF
		Rcp.cmd_RcpOperation := 10;
		RCP.Pause_ET := T#0S;
END_CASE
RCP.iRcpStepN := nRcpIndex;

END_PROGRAM

// ---- POUs/FB_RecipeAnalogControlInputSequencer.TcPOU
FUNCTION_BLOCK FB_RecipeAnalogControlInputSequencer
VAR_INPUT
	tempRecipe: REAL;
	pressRecipe: REAL;
	rotRecipe: REAL;
	rampTime: UINT;
END_VAR
VAR_IN_OUT
	rRecipe: ARRAY[1..26] OF REAL;
END_VAR
VAR
	i: UINT;
END_VAR

FOR i:= 1 TO 26 DO
	GVL_IO.aController[i].input.restart := TRUE;
	GVL_IO.aController[i].input.rampTime := rampTime; 
	GVL_IO.aController[i].input.targetValue := rRecipe[i];
END_FOR

GVL_IO.aController[27].input.restart := TRUE;
GVL_IO.aController[27].input.rampTime := rampTime;
GVL_IO.aController[27].input.targetValue := tempRecipe;

GVL_IO.aController[28].input.restart := TRUE;
GVL_IO.aController[28].input.rampTime := rampTime;
GVL_IO.aController[28].input.targetValue := pressRecipe;

GVL_IO.aController[29].input.restart := TRUE;
GVL_IO.aController[29].input.rampTime := rampTime;
GVL_IO.aController[29].input.targetValue := rotRecipe;

END_FUNCTION_BLOCK

// ---- POUs/FB_ValveControl.TcPOU
FUNCTION_BLOCK FB_ValveControl
VAR_INPUT
	valveSetting: DWORD; 
END_VAR

(* Solenoid Valve Mapping *)
GVL_IO.aOutputSolValve[1].0 := valveSetting.0; //V01 Hyd. Carrier
GVL_IO.aOutputSolValve[1].1 := valveSetting.1; //V02
GVL_IO.aOutputSolValve[1].2 := valveSetting.2; //V03
GVL_IO.aOutputSolValve[1].3 := valveSetting.3; //V04
GVL_IO.aOutputSolValve[1].4 := valveSetting.4; //V05
GVL_IO.aOutputSolValve[1].6 := valveSetting.5; //V07
GVL_IO.aOutputSolValve[1].7 := valveSetting.6; //V08
GVL_IO.aOutputSolValve[1].9 := valveSetting.7; //V10
GVL_IO.aOutputSolValve[1].10 := valveSetting.8; //V11
GVL_IO.aOutputSolValve[1].12 := valveSetting.9; //V13
GVL_IO.aOutputSolValve[1].13 := valveSetting.10; //V14
GVL_IO.aOutputSolValve[1].15 := valveSetting.11; //V16
GVL_IO.aOutputSolValve[2].0 := valveSetting.12; //V17
GVL_IO.aOutputSolValve[2].2 := valveSetting.13; //V19
GVL_IO.aOutputSolValve[2].3 := valveSetting.14; //V20
GVL_IO.aOutputSolValve[2].5 := valveSetting.15; //V22
GVL_IO.aOutputSolValve[2].6 := valveSetting.16; //V23
GVL_IO.aOutputSolValve[2].7 := valveSetting.17; //V24
GVL_IO.aOutputSolValve[2].8 := valveSetting.18; //V25
GVL_IO.aOutputSolValve[2].9 := valveSetting.19; //V26
GVL_IO.aOutputSolValve[2].10 := valveSetting.20; //V27
GVL_IO.aOutputSolValve[2].11 := valveSetting.21; //V28
GVL_IO.aOutputSolValve[2].12 := valveSetting.22; //V29
GVL_IO.aOutputSolValve[2].13 := valveSetting.23; //V30
GVL_IO.aOutputSolValve[2].14 := valveSetting.24; //V31
GVL_IO.aOutputSolValve[2].15 := valveSetting.25; //V32

END_FUNCTION_BLOCK

// ---- POUs/FB_TON_Pausable.TcPOU
FUNCTION_BLOCK FB_TON_Pausable
VAR_INPUT
	IN      : BOOL;     (* Start/Stop the timer *)
    PT      : TIME;     (* Preset time *)
    PAUSE   : BOOL;     (* Pause the timer *)
END_VAR
VAR_OUTPUT
	Q       : BOOL;     (* Output: TRUE when PT is reached *)
    ET      : TIME;     (* Elapsed time *)
END_VAR
VAR
	// Internal variables
    fbTON   : TON;      (* Standard TON to do the actual timing when not paused *)
    tElapsedAtPause : TIME; (* Stores ET when paused *)
    bWasPaused      : BOOL; (* Helps detect the rising edge of PAUSE *)
    bOldIn          : BOOL; (* Stores previous IN state for rising/falling edge detection *)
END_VAR

IF NOT IN THEN
    // Reset condition: IN is FALSE
    tElapsedAtPause := T#0S;
    ET := T#0S;
    Q := FALSE;
    fbTON(IN := FALSE); // Ensure internal TON is also reset
    bWasPaused := FALSE; // Reset pause state
ELSIF IN THEN
    // Timer is active
    IF PAUSE THEN
        // PAUSE is active
        IF NOT bWasPaused THEN
            // Rising edge of PAUSE: Capture current elapsed time from TON
            tElapsedAtPause := tElapsedAtPause + fbTON.ET;
            bWasPaused := TRUE;
        END_IF
        // Timer is paused: ET does not advance
        ET := tElapsedAtPause;
        Q := (ET >= PT); // Q remains based on the paused ET
        fbTON(IN := FALSE); // Stop the internal TON from running
    ELSE (* NOT PAUSE *)
        // PAUSE is not active, run the timer
        bWasPaused := FALSE; // Clear paused state

        // Adjust PT for the internal TON to account for time spent paused
        // Only call TON if IN is TRUE and NOT PAUSE
        fbTON(
            IN := TRUE,
            PT := PT - tElapsedAtPause (* Subtract time already elapsed/paused *)
        );

        // Calculate actual ET for output
        // It's the time accumulated before pause + time accumulated after resume
        ET := tElapsedAtPause + fbTON.ET;
        Q := fbTON.Q;
    END_IF
END_IF

// Store current IN state for next cycle's edge detection
bOldIn := IN;

END_FUNCTION_BLOCK

// ---- POUs/F_ResetTimersAndRCPTimes.TcPOU
FUNCTION F_ResetTimersAndRCPTimes : BOOL
VAR_IN_OUT // These are references to the actual TON instances and the RCP structure
    fbPause_TON : TON;
    fbRamp_TON  : FB_TON_Pausable;
    fbHold_TON  : FB_TON_Pausable;
END_VAR

// Reset the timers by setting IN to FALSE
fbPause_TON(IN:=FALSE); // Calling the TON FB instances
fbRamp_TON(IN:=FALSE, Pause:=FALSE);
fbHold_TON(IN:=FALSE, Pause:=FALSE);

// Reset the elapsed times in the RCP structure
RCP.Pause_ET := T#0S;
RCP.RecipeRunET.ET := T#0S;
RCP.RecipeRunET.Mode := E_RecipeRunETMode.None;

F_ResetTimersAndRCPTimes := TRUE; // Indicate successful execution (optional)

END_FUNCTION

// ---- POUs/P31_PriorityControl.TcPOU
PROGRAM P31_PriorityControl
VAR
	fbAnalogDeviceRampControl : FB_AnalogDeviceRampControl;
	i : UINT;
END_VAR
VAR_OUTPUT
	complete : BOOL;
END_VAR

fbAnalogDeviceRampControl();
complete := TRUE;
FOR i := 1 TO GVL_IO.NumAnalogController DO
	IF GVL_IO.aController[i].targetValueReached = FALSE THEN
		complete := FALSE;
		EXIT;
	END_IF
END_FOR

END_PROGRAM

// ---- POUs/P60_UpdatePV.TcPOU
PROGRAM P60_UpdatePV
VAR
	i: UINT;
END_VAR

FOR i:=1 TO GVL_IO.NumFlowController DO
	GVL_IO.aController_PV[i] := (INT_TO_REAL(GVL_IO.aAnalogInputIO[i]) / GVL_IO.KL3464MaxValueH) * GVL_IO.AnalogControllerOutputVoltage;
END_FOR

GVL_IO.aController_PV[27] := WORD_TO_REAL(GVL_IO.wE3508_PV);
GVL_IO.aController_PV[28] := WORD_TO_REAL(GVL_IO.wIqPlus_CDG2_PV);
GVL_IO.aController_PV[29] := GVL_IO.nRotation_Converted_PV;

END_PROGRAM

